LIN {X -0.088,Y -488.926,Z 1104.794,A 0.000,B 0.000,C 90.000,E1 358.969} C_DIS
LIN {X 0.190,Y -496.704,Z 1104.791,A 0.000,B 0.000,C 90.000,E1 358.396} C_DIS
LIN {X -0.080,Y -504.149,Z 1104.788,A 0.000,B 0.000,C 90.000,E1 357.879} C_DIS
LIN {X 0.232,Y -511.620,Z 1104.785,A 0.000,B 0.000,C 90.000,E1 357.249} C_DIS
LIN {X 0.051,Y -516.072,Z 1104.783,A 0.000,B 0.000,C 90.000,E1 356.906} C_DIS
LIN {X 0.077,Y -522.941,Z 1104.779,A 0.000,B 0.000,C 90.000,E1 356.274} C_DIS
LIN {X -0.241,Y -529.630,Z 1104.776,A 0.000,B 0.000,C 90.000,E1 355.641} C_DIS
LIN {X 0.250,Y -535.894,Z 1104.772,A 0.000,B 0.000,C 90.000,E1 354.894} C_DIS
LIN {X -0.207,Y -540.523,Z 1104.769,A 0.000,B 0.000,C 90.000,E1 354.375} C_DIS
LIN {X 0.140,Y -545.729,Z 1104.765,A 0.000,B 0.000,C 90.000,E1 353.628} C_DIS
LIN {X 0.057,Y -550.505,Z 1104.761,A 0.000,B 0.000,C 90.000,E1 352.932} C_DIS
LIN {X 0.201,Y -554.018,Z 1104.758,A 0.000,B 0.000,C 90.000,E1 352.356} C_DIS
LIN {X 0.196,Y -557.831,Z 1104.754,A 0.000,B 0.000,C 90.000,E1 351.659} C_DIS
LIN {X 0.142,Y -561.247,Z 1104.750,A 0.000,B 0.000,C 90.000,E1 350.971} C_DIS
LIN {X 0.135,Y -563.191,Z 1104.748,A 0.000,B 0.000,C 90.000,E1 350.557} C_DIS
LIN {X -0.033,Y -566.692,Z 1104.743,A 0.000,B 0.000,C 90.000,E1 349.746} C_DIS
LIN {X -0.067,Y -569.959,Z 1104.739,A 0.000,B 0.000,C 90.000,E1 348.926} C_DIS
LIN {X 0.014,Y -574.006,Z 1104.732,A 0.000,B 0.000,C 90.000,E1 347.825} C_DIS
LIN {X 0.183,Y -576.822,Z 1104.728,A 0.000,B 0.000,C 90.000,E1 346.992} C_DIS
LIN {X 0.132,Y -581.130,Z 1104.720,A 0.000,B 0.000,C 90.000,E1 345.644} C_DIS
LIN {X 0.059,Y -584.388,Z 1104.714,A 0.000,B 0.000,C 90.000,E1 344.574} C_DIS
LIN {X -0.293,Y -588.324,Z 1104.707,A 0.000,B 0.000,C 90.000,E1 343.268} C_DIS
LIN {X 0.148,Y -592.034,Z 1104.700,A 0.000,B 0.000,C 90.000,E1 341.891} C_DIS
LIN {X -0.166,Y -594.797,Z 1104.694,A 0.000,B 0.000,C 90.000,E1 340.859} C_DIS
LIN {X 0.323,Y -597.309,Z 1104.688,A 0.000,B 0.000,C 90.000,E1 339.752} C_DIS
LIN {X -0.004,Y -600.116,Z 1104.680,A 0.000,B 0.000,C 90.000,E1 338.465} C_DIS
LIN {X 0.086,Y -601.519,Z 1104.676,A 0.000,B 0.000,C 90.000,E1 337.667} C_DIS
LIN {X 0.187,Y -602.833,Z 1104.672,A 0.000,B 0.000,C 90.000,E1 336.869} C_DIS
LIN {X -0.015,Y -603.928,Z 1104.667,A 0.000,B 0.000,C 90.000,E1 336.102} C_DIS
LIN {X 0.042,Y -605.238,Z 1104.661,A 0.000,B 0.000,C 90.000,E1 335.049} C_DIS
LIN {X -0.235,Y -606.531,Z 1104.654,A 0.000,B 0.000,C 90.000,E1 333.768} C_DIS
LIN {X 0.153,Y -607.021,Z 1104.650,A 0.000,B 0.000,C 90.000,E1 332.948} C_DIS
LIN {X 0.284,Y -607.391,Z 1104.646,A 0.000,B 0.000,C 90.000,E1 332.153} C_DIS
LIN {X 0.086,Y -607.526,Z 1104.640,A 0.000,B 0.000,C 90.000,E1 331.129} C_DIS
LIN {X 0.281,Y -607.417,Z 1104.637,A 0.000,B 0.000,C 90.000,E1 330.589} C_DIS
LIN {X -0.151,Y -606.764,Z 1104.631,A 0.000,B 0.000,C 90.000,E1 329.587} C_DIS
LIN {X -0.010,Y -605.795,Z 1104.627,A 0.000,B 0.000,C 90.000,E1 328.791} C_DIS
LIN {X 0.047,Y -604.102,Z 1104.621,A 0.000,B 0.000,C 90.000,E1 327.740} C_DIS
LIN {X -0.032,Y -602.427,Z 1104.616,A 0.000,B 0.000,C 90.000,E1 326.962} C_DIS
LIN {X 0.291,Y -599.833,Z 1104.611,A 0.000,B 0.000,C 90.000,E1 325.881} C_DIS
LIN {X -0.182,Y -596.179,Z 1104.603,A 0.000,B 0.000,C 90.000,E1 324.609} C_DIS
LIN {X -0.016,Y -591.507,Z 1104.594,A 0.000,B 0.000,C 90.000,E1 323.004} C_DIS
LIN {X 0.146,Y -589.181,Z 1104.590,A 0.000,B 0.000,C 90.000,E1 322.190} C_DIS
LIN {X -0.149,Y -585.017,Z 1104.583,A 0.000,B 0.000,C 90.000,E1 320.884} C_DIS
LIN {X -0.050,Y -582.539,Z 1104.578,A 0.000,B 0.000,C 90.000,E1 320.070} C_DIS
LIN {X -0.256,Y -578.919,Z 1104.572,A 0.000,B 0.000,C 90.000,E1 319.013} C_DIS
LIN {X 0.156,Y -575.977,Z 1104.568,A 0.000,B 0.000,C 90.000,E1 318.162} C_DIS
LIN {X -0.276,Y -572.557,Z 1104.563,A 0.000,B 0.000,C 90.000,E1 317.391} C_DIS
LIN {X -0.192,Y -569.234,Z 1104.559,A 0.000,B 0.000,C 90.000,E1 316.701} C_DIS
LIN {X 0.004,Y -566.303,Z 1104.556,A 0.000,B 0.000,C 90.000,E1 316.134} C_DIS
LIN {X 0.024,Y -562.362,Z 1104.552,A 0.000,B 0.000,C 90.000,E1 315.445} C_DIS
LIN {X -0.331,Y -556.410,Z 1104.547,A 0.000,B 0.000,C 90.000,E1 314.514} C_DIS
LIN {X -0.008,Y -551.946,Z 1104.543,A 0.000,B 0.000,C 90.000,E1 313.785} C_DIS
LIN {X -0.110,Y -547.705,Z 1104.539,A 0.000,B 0.000,C 90.000,E1 313.095} C_DIS
LIN {X 0.148,Y -541.824,Z 1104.534,A 0.000,B 0.000,C 90.000,E1 312.081} C_DIS
LIN {X -0.036,Y -538.515,Z 1104.530,A 0.000,B 0.000,C 90.000,E1 311.391} C_DIS
LIN {X 0.013,Y -535.602,Z 1104.525,A 0.000,B 0.000,C 90.000,E1 310.458} C_DIS
LIN {X 0.015,Y -534.100,Z 1104.520,A 0.000,B 0.000,C 90.000,E1 309.600} C_DIS
LIN {X -0.229,Y -533.704,Z 1104.519,A 0.000,B 0.000,C 90.000,E1 309.483} C_DIS
LIN {X -0.071,Y -532.956,Z 1104.516,A 0.000,B 0.000,C 90.000,E1 308.830} C_DIS
LIN {X 0.219,Y -532.151,Z 1104.508,A 0.000,B 0.000,C 90.000,E1 307.363} C_DIS
LIN {X 0.191,Y -532.113,Z 1104.503,A 0.000,B 0.000,C 90.000,E1 306.503} C_DIS
LIN {X 0.171,Y -532.219,Z 1104.500,A 0.000,B 0.000,C 90.000,E1 305.931} C_DIS
LIN {X -0.085,Y -533.150,Z 1104.485,A 0.000,B 0.000,C 90.000,E1 303.372} C_DIS
LIN {X -0.145,Y -534.752,Z 1104.471,A 0.000,B 0.000,C 90.000,E1 300.797} C_DIS
LIN {X 0.175,Y -535.550,Z 1104.465,A 0.000,B 0.000,C 90.000,E1 299.617} C_DIS
LIN {X 0.040,Y -536.287,Z 1104.458,A 0.000,B 0.000,C 90.000,E1 298.487} C_DIS
LIN {X 0.028,Y -537.260,Z 1104.447,A 0.000,B 0.000,C 90.000,E1 296.488} C_DIS
LIN {X -0.142,Y -537.865,Z 1104.439,A 0.000,B 0.000,C 90.000,E1 295.079} C_DIS
LIN {X -0.042,Y -538.253,Z 1104.431,A 0.000,B 0.000,C 90.000,E1 293.643} C_DIS
LIN {X 0.068,Y -538.548,Z 1104.423,A 0.000,B 0.000,C 90.000,E1 292.206} C_DIS
LIN {X -0.246,Y -538.753,Z 1104.417,A 0.000,B 0.000,C 90.000,E1 291.099} C_DIS
LIN {X -0.053,Y -538.752,Z 1104.411,A 0.000,B 0.000,C 90.000,E1 289.939} C_DIS
LIN {X 0.185,Y -538.574,Z 1104.403,A 0.000,B 0.000,C 90.000,E1 288.489} C_DIS
LIN {X -0.096,Y -538.268,Z 1104.395,A 0.000,B 0.000,C 90.000,E1 287.094} C_DIS
LIN {X -0.089,Y -537.971,Z 1104.389,A 0.000,B 0.000,C 90.000,E1 285.953} C_DIS
LIN {X -0.178,Y -537.394,Z 1104.381,A 0.000,B 0.000,C 90.000,E1 284.537} C_DIS
LIN {X -0.211,Y -536.591,Z 1104.371,A 0.000,B 0.000,C 90.000,E1 282.827} C_DIS
LIN {X 0.149,Y -535.751,Z 1104.362,A 0.000,B 0.000,C 90.000,E1 281.074} C_DIS
LIN {X -0.042,Y -534.871,Z 1104.352,A 0.000,B 0.000,C 90.000,E1 279.378} C_DIS
LIN {X 0.096,Y -534.050,Z 1104.343,A 0.000,B 0.000,C 90.000,E1 277.644} C_DIS
LIN {X 0.218,Y -533.208,Z 1104.333,A 0.000,B 0.000,C 90.000,E1 275.910} C_DIS
LIN {X 0.230,Y -532.560,Z 1104.325,A 0.000,B 0.000,C 90.000,E1 274.473} C_DIS
LIN {X 0.201,Y -531.620,Z 1104.314,A 0.000,B 0.000,C 90.000,E1 272.465} C_DIS
LIN {X 0.140,Y -530.818,Z 1104.304,A 0.000,B 0.000,C 90.000,E1 270.745} C_DIS
LIN {X 0.051,Y -529.984,Z 1104.295,A 0.000,B 0.000,C 90.000,E1 269.026} C_DIS
LIN {X -0.025,Y -529.212,Z 1104.287,A 0.000,B 0.000,C 90.000,E1 267.593} C_DIS
LIN {X -0.138,Y -527.983,Z 1104.275,A 0.000,B 0.000,C 90.000,E1 265.584} C_DIS
LIN {X -0.182,Y -527.252,Z 1104.269,A 0.000,B 0.000,C 90.000,E1 264.432} C_DIS
LIN {X -0.249,Y -526.568,Z 1104.264,A 0.000,B 0.000,C 90.000,E1 263.571} C_DIS
LIN {X 0.268,Y -525.419,Z 1104.258,A 0.000,B 0.000,C 90.000,E1 262.356} C_DIS
LIN {X 0.215,Y -523.033,Z 1104.245,A 0.000,B 0.000,C 90.000,E1 260.038} C_DIS
LIN {X 0.253,Y -521.957,Z 1104.238,A 0.000,B 0.000,C 90.000,E1 258.870} C_DIS
LIN {X -0.229,Y -519.974,Z 1104.227,A 0.000,B 0.000,C 90.000,E1 256.881} C_DIS
LIN {X -0.130,Y -518.620,Z 1104.219,A 0.000,B 0.000,C 90.000,E1 255.408} C_DIS
LIN {X 0.072,Y -517.057,Z 1104.211,A 0.000,B 0.000,C 90.000,E1 253.921} C_DIS
LIN {X 0.148,Y -516.161,Z 1104.206,A 0.000,B 0.000,C 90.000,E1 253.032} C_DIS
LIN {X 0.081,Y -514.287,Z 1104.196,A 0.000,B 0.000,C 90.000,E1 251.275} C_DIS
LIN {X -0.084,Y -513.016,Z 1104.190,A 0.000,B 0.000,C 90.000,E1 250.115} C_DIS
LIN {X -0.031,Y -510.937,Z 1104.180,A 0.000,B 0.000,C 90.000,E1 248.337} C_DIS
LIN {X 0.055,Y -509.197,Z 1104.172,A 0.000,B 0.000,C 90.000,E1 246.847} C_DIS
LIN {X 0.101,Y -506.997,Z 1104.163,A 0.000,B 0.000,C 90.000,E1 245.357} C_DIS
LIN {X 0.134,Y -505.675,Z 1104.158,A 0.000,B 0.000,C 90.000,E1 244.460} C_DIS
LIN {X 0.235,Y -503.739,Z 1104.152,A 0.000,B 0.000,C 90.000,E1 243.256} C_DIS
LIN {X -0.232,Y -500.810,Z 1104.142,A 0.000,B 0.000,C 90.000,E1 241.513} C_DIS
LIN {X 0.155,Y -497.771,Z 1104.132,A 0.000,B 0.000,C 90.000,E1 239.665} C_DIS
LIN {X 0.174,Y -495.736,Z 1104.125,A 0.000,B 0.000,C 90.000,E1 238.456} C_DIS
LIN {X 0.275,Y -492.520,Z 1104.115,A 0.000,B 0.000,C 90.000,E1 236.628} C_DIS
LIN {X -0.204,Y -490.375,Z 1104.108,A 0.000,B 0.000,C 90.000,E1 235.468} C_DIS
LIN {X 0.081,Y -487.511,Z 1104.100,A 0.000,B 0.000,C 90.000,E1 233.909} C_DIS
LIN {X -0.075,Y -484.603,Z 1104.091,A 0.000,B 0.000,C 90.000,E1 232.396} C_DIS
LIN {X 0.017,Y -481.539,Z 1104.083,A 0.000,B 0.000,C 90.000,E1 230.848} C_DIS
LIN {X -0.044,Y -477.231,Z 1104.071,A 0.000,B 0.000,C 90.000,E1 228.690} C_DIS
LIN {X -0.176,Y -472.439,Z 1104.057,A 0.000,B 0.000,C 90.000,E1 226.215} C_DIS
LIN {X -0.057,Y -469.619,Z 1104.048,A 0.000,B 0.000,C 90.000,E1 224.636} C_DIS
LIN {X -0.067,Y -467.362,Z 1104.041,A 0.000,B 0.000,C 90.000,E1 223.380} C_DIS
LIN {X 0.104,Y -463.361,Z 1104.029,A 0.000,B 0.000,C 90.000,E1 221.148} C_DIS
LIN {X 0.218,Y -459.609,Z 1104.016,A 0.000,B 0.000,C 90.000,E1 218.910} C_DIS
LIN {X -0.068,Y -456.459,Z 1104.006,A 0.000,B 0.000,C 90.000,E1 217.030} C_DIS
LIN {X -0.060,Y -453.498,Z 1103.995,A 0.000,B 0.000,C 90.000,E1 215.105} C_DIS
LIN {X 0.069,Y -450.030,Z 1103.983,A 0.000,B 0.000,C 90.000,E1 212.832} C_DIS
LIN {X 0.169,Y -447.237,Z 1103.972,A 0.000,B 0.000,C 90.000,E1 210.875} C_DIS
LIN {X -0.014,Y -443.021,Z 1103.954,A 0.000,B 0.000,C 90.000,E1 207.641} C_DIS
LIN {X 0.091,Y -440.560,Z 1103.941,A 0.000,B 0.000,C 90.000,E1 205.335} C_DIS
LIN {X 0.076,Y -439.566,Z 1103.932,A 0.000,B 0.000,C 90.000,E1 203.695} C_DIS
LIN {X 0.024,Y -439.516,Z 1103.924,A 0.000,B 0.000,C 90.000,E1 202.386} C_DIS
LIN {X -0.037,Y -440.005,Z 1103.919,A 0.000,B 0.000,C 90.000,E1 201.408} C_DIS
LIN {X 0.065,Y -440.657,Z 1103.915,A 0.000,B 0.000,C 90.000,E1 200.737} C_DIS
LIN {X 0.174,Y -441.671,Z 1103.912,A 0.000,B 0.000,C 90.000,E1 200.066} C_DIS
LIN {X 0.142,Y -443.785,Z 1103.906,A 0.000,B 0.000,C 90.000,E1 199.087} C_DIS
LIN {X -0.010,Y -446.435,Z 1103.901,A 0.000,B 0.000,C 90.000,E1 198.127} C_DIS
LIN {X 0.040,Y -451.871,Z 1103.892,A 0.000,B 0.000,C 90.000,E1 196.496} C_DIS
LIN {X -0.008,Y -464.587,Z 1103.874,A 0.000,B 0.000,C 90.000,E1 193.300} C_DIS
LIN {X 0.197,Y -476.298,Z 1103.859,A 0.000,B 0.000,C 90.000,E1 190.602} C_DIS
LIN {X -0.165,Y -483.419,Z 1103.850,A 0.000,B 0.000,C 90.000,E1 189.095} C_DIS
LIN {X -0.062,Y -489.809,Z 1103.843,A 0.000,B 0.000,C 90.000,E1 187.701} C_DIS
LIN {X -0.243,Y -496.743,Z 1103.834,A 0.000,B 0.000,C 90.000,E1 186.201} C_DIS
LIN {X 0.077,Y -504.800,Z 1103.824,A 0.000,B 0.000,C 90.000,E1 184.359} C_DIS
LIN {X 0.126,Y -511.555,Z 1103.816,A 0.000,B 0.000,C 90.000,E1 182.865} C_DIS
LIN {X -0.079,Y -520.276,Z 1103.805,A 0.000,B 0.000,C 90.000,E1 180.974} C_DIS
LIN {X 0.222,Y -527.050,Z 1103.797,A 0.000,B 0.000,C 90.000,E1 179.484} C_DIS
LIN {X 0.135,Y -533.740,Z 1103.789,A 0.000,B 0.000,C 90.000,E1 178.051} C_DIS
LIN {X -0.103,Y -539.767,Z 1103.782,A 0.000,B 0.000,C 90.000,E1 176.788} C_DIS
LIN {X 0.007,Y -545.093,Z 1103.776,A 0.000,B 0.000,C 90.000,E1 175.641} C_DIS
LIN {X -0.169,Y -552.915,Z 1103.766,A 0.000,B 0.000,C 90.000,E1 173.970} C_DIS
LIN {X 0.065,Y -560.117,Z 1103.758,A 0.000,B 0.000,C 90.000,E1 172.413} C_DIS
LIN {X -0.052,Y -565.284,Z 1103.752,A 0.000,B 0.000,C 90.000,E1 171.319} C_DIS
LIN {X -0.162,Y -570.987,Z 1103.745,A 0.000,B 0.000,C 90.000,E1 170.095} C_DIS
LIN {X -0.199,Y -578.362,Z 1103.736,A 0.000,B 0.000,C 90.000,E1 168.465} C_DIS
LIN {X -0.218,Y -584.227,Z 1103.728,A 0.000,B 0.000,C 90.000,E1 167.117} C_DIS
LIN {X 0.320,Y -588.658,Z 1103.722,A 0.000,B 0.000,C 90.000,E1 165.992} C_DIS
LIN {X 0.206,Y -592.896,Z 1103.716,A 0.000,B 0.000,C 90.000,E1 164.936} C_DIS
LIN {X -0.276,Y -596.934,Z 1103.711,A 0.000,B 0.000,C 90.000,E1 163.921} C_DIS
LIN {X 0.044,Y -600.692,Z 1103.705,A 0.000,B 0.000,C 90.000,E1 162.834} C_DIS
LIN {X 0.240,Y -604.257,Z 1103.699,A 0.000,B 0.000,C 90.000,E1 161.764} C_DIS
LIN {X -0.180,Y -608.308,Z 1103.692,A 0.000,B 0.000,C 90.000,E1 160.496} C_DIS
LIN {X -0.062,Y -611.408,Z 1103.686,A 0.000,B 0.000,C 90.000,E1 159.444} C_DIS
LIN {X -0.114,Y -614.384,Z 1103.680,A 0.000,B 0.000,C 90.000,E1 158.411} C_DIS
LIN {X 0.073,Y -617.924,Z 1103.673,A 0.000,B 0.000,C 90.000,E1 157.102} C_DIS
LIN {X 0.320,Y -622.024,Z 1103.664,A 0.000,B 0.000,C 90.000,E1 155.537} C_DIS
LIN {X 0.079,Y -625.940,Z 1103.656,A 0.000,B 0.000,C 90.000,E1 154.024} C_DIS
LIN {X 0.161,Y -629.006,Z 1103.649,A 0.000,B 0.000,C 90.000,E1 152.743} C_DIS
LIN {X -0.238,Y -632.386,Z 1103.640,A 0.000,B 0.000,C 90.000,E1 151.257} C_DIS
LIN {X -0.271,Y -635.740,Z 1103.632,A 0.000,B 0.000,C 90.000,E1 149.744} C_DIS
LIN {X 0.042,Y -638.341,Z 1103.625,A 0.000,B 0.000,C 90.000,E1 148.456} C_DIS
LIN {X 0.064,Y -640.833,Z 1103.618,A 0.000,B 0.000,C 90.000,E1 147.199} C_DIS
LIN {X -0.077,Y -643.237,Z 1103.611,A 0.000,B 0.000,C 90.000,E1 145.960} C_DIS
LIN {X -0.227,Y -645.049,Z 1103.605,A 0.000,B 0.000,C 90.000,E1 144.975} C_DIS
LIN {X -0.018,Y -647.746,Z 1103.597,A 0.000,B 0.000,C 90.000,E1 143.463} C_DIS
LIN {X -0.142,Y -650.395,Z 1103.589,A 0.000,B 0.000,C 90.000,E1 141.984} C_DIS
LIN {X 0.105,Y -653.631,Z 1103.579,A 0.000,B 0.000,C 90.000,E1 140.231} C_DIS
LIN {X 0.306,Y -657.423,Z 1103.568,A 0.000,B 0.000,C 90.000,E1 138.243} C_DIS
LIN {X 0.170,Y -660.396,Z 1103.560,A 0.000,B 0.000,C 90.000,E1 136.782} C_DIS
LIN {X 0.033,Y -665.717,Z 1103.547,A 0.000,B 0.000,C 90.000,E1 134.352} C_DIS
LIN {X 0.081,Y -670.402,Z 1103.536,A 0.000,B 0.000,C 90.000,E1 132.405} C_DIS
LIN {X -0.296,Y -674.041,Z 1103.528,A 0.000,B 0.000,C 90.000,E1 130.987} C_DIS
LIN {X -0.025,Y -677.589,Z 1103.520,A 0.000,B 0.000,C 90.000,E1 129.519} C_DIS
LIN {X 0.356,Y -681.922,Z 1103.510,A 0.000,B 0.000,C 90.000,E1 127.810} C_DIS
LIN {X -0.206,Y -684.985,Z 1103.504,A 0.000,B 0.000,C 90.000,E1 126.664} C_DIS
LIN {X -0.137,Y -688.563,Z 1103.496,A 0.000,B 0.000,C 90.000,E1 125.231} C_DIS
LIN {X -0.049,Y -691.400,Z 1103.489,A 0.000,B 0.000,C 90.000,E1 124.040} C_DIS
LIN {X -0.302,Y -694.311,Z 1103.483,A 0.000,B 0.000,C 90.000,E1 122.880} C_DIS
LIN {X -0.162,Y -696.602,Z 1103.477,A 0.000,B 0.000,C 90.000,E1 121.926} C_DIS
LIN {X -0.357,Y -698.662,Z 1103.472,A 0.000,B 0.000,C 90.000,E1 121.003} C_DIS
LIN {X -0.168,Y -700.440,Z 1103.467,A 0.000,B 0.000,C 90.000,E1 120.050} C_DIS
LIN {X -0.042,Y -702.354,Z 1103.460,A 0.000,B 0.000,C 90.000,E1 118.871} C_DIS
LIN {X 0.121,Y -703.558,Z 1103.455,A 0.000,B 0.000,C 90.000,E1 117.924} C_DIS
LIN {X -0.273,Y -704.299,Z 1103.451,A 0.000,B 0.000,C 90.000,E1 117.257} C_DIS
LIN {X -0.124,Y -705.370,Z 1103.444,A 0.000,B 0.000,C 90.000,E1 115.848} C_DIS
LIN {X -0.194,Y -705.737,Z 1103.440,A 0.000,B 0.000,C 90.000,E1 115.155} C_DIS
LIN {X 0.387,Y -705.696,Z 1103.437,A 0.000,B 0.000,C 90.000,E1 114.643} C_DIS
LIN {X -0.258,Y -705.486,Z 1103.436,A 0.000,B 0.000,C 90.000,E1 114.463} C_DIS
LIN {X 0.319,Y -704.770,Z 1103.433,A 0.000,B 0.000,C 90.000,E1 113.951} C_DIS
LIN {X -0.040,Y -703.023,Z 1103.431,A 0.000,B 0.000,C 90.000,E1 113.515} C_DIS
LIN {X 0.239,Y -701.954,Z 1103.429,A 0.000,B 0.000,C 90.000,E1 113.259} C_DIS
LIN {X -0.033,Y -698.059,Z 1103.427,A 0.000,B 0.000,C 90.000,E1 112.823} C_DIS
LIN {X 0.096,Y -696.956,Z 1103.426,A 0.000,B 0.000,C 90.000,E1 112.695} C_DIS
LIN {X -0.042,Y -695.323,Z 1103.426,A 0.000,B 0.000,C 90.000,E1 112.589} C_DIS
LIN {X -0.005,Y -690.723,Z 1103.424,A 0.000,B 0.000,C 90.000,E1 112.386} C_DIS
LIN {X -0.108,Y -687.387,Z 1103.424,A 0.000,B 0.000,C 90.000,E1 112.259} C_DIS
LIN {X -0.283,Y -685.495,Z 1103.423,A 0.000,B 0.000,C 90.000,E1 112.206} C_DIS
LIN {X -0.053,Y -683.590,Z 1103.423,A 0.000,B 0.000,C 90.000,E1 112.153} C_DIS
LIN {X -0.199,Y -675.939,Z 1103.423,A 0.000,B 0.000,C 90.000,E1 112.078} C_DIS
LIN {X -0.225,Y -604.098,Z 1103.423,A 0.000,B 0.000,C 90.000,E1 112.078} C_DIS
LIN {X 0.135,Y -600.461,Z 1103.422,A 0.000,B 0.000,C 90.000,E1 111.844} C_DIS
LIN {X 0.160,Y -596.106,Z 1103.420,A 0.000,B 0.000,C 90.000,E1 111.535} C_DIS
LIN {X -0.062,Y -578.609,Z 1103.411,A 0.000,B 0.000,C 90.000,E1 110.066} C_DIS
LIN {X -0.014,Y -574.362,Z 1103.410,A 0.000,B 0.000,C 90.000,E1 109.704} C_DIS
LIN {X -0.171,Y -568.294,Z 1103.407,A 0.000,B 0.000,C 90.000,E1 109.268} C_DIS
LIN {X 0.173,Y -560.101,Z 1103.404,A 0.000,B 0.000,C 90.000,E1 108.725} C_DIS
LIN {X 0.117,Y -553.768,Z 1103.402,A 0.000,B 0.000,C 90.000,E1 108.362} C_DIS
LIN {X 0.221,Y -549.835,Z 1103.401,A 0.000,B 0.000,C 90.000,E1 108.055} C_DIS
LIN {X 0.135,Y -548.522,Z 1103.399,A 0.000,B 0.000,C 90.000,E1 107.873} C_DIS
LIN {X 0.094,Y -548.497,Z 1103.399,A 0.000,B 0.000,C 90.000,E1 107.873} C_DIS
LIN {X 0.224,Y -548.201,Z 1103.398,A 0.000,B 0.000,C 90.000,E1 107.583} C_DIS
LIN {X 0.264,Y -548.501,Z 1103.393,A 0.000,B 0.000,C 90.000,E1 106.677} C_DIS
LIN {X -0.234,Y -550.066,Z 1103.380,A 0.000,B 0.000,C 90.000,E1 104.481} C_DIS
LIN {X -0.284,Y -551.856,Z 1103.368,A 0.000,B 0.000,C 90.000,E1 102.243} C_DIS
LIN {X -0.107,Y -553.448,Z 1103.359,A 0.000,B 0.000,C 90.000,E1 100.546} C_DIS
LIN {X 0.126,Y -555.451,Z 1103.348,A 0.000,B 0.000,C 90.000,E1 98.568} C_DIS
LIN {X 0.060,Y -556.875,Z 1103.340,A 0.000,B 0.000,C 90.000,E1 97.182} C_DIS
LIN {X -0.108,Y -558.046,Z 1103.334,A 0.000,B 0.000,C 90.000,E1 96.087} C_DIS
LIN {X -0.260,Y -559.127,Z 1103.328,A 0.000,B 0.000,C 90.000,E1 94.992} C_DIS
LIN {X 0.241,Y -560.227,Z 1103.320,A 0.000,B 0.000,C 90.000,E1 93.555} C_DIS
LIN {X 0.167,Y -561.129,Z 1103.312,A 0.000,B 0.000,C 90.000,E1 92.178} C_DIS
LIN {X 0.206,Y -562.026,Z 1103.303,A 0.000,B 0.000,C 90.000,E1 90.516} C_DIS
LIN {X -0.054,Y -562.417,Z 1103.298,A 0.000,B 0.000,C 90.000,E1 89.714} C_DIS
LIN {X -0.108,Y -563.095,Z 1103.291,A 0.000,B 0.000,C 90.000,E1 88.339} C_DIS
LIN {X -0.006,Y -563.848,Z 1103.282,A 0.000,B 0.000,C 90.000,E1 86.674} C_DIS
LIN {X 0.121,Y -564.536,Z 1103.272,A 0.000,B 0.000,C 90.000,E1 85.008} C_DIS
LIN {X 0.154,Y -565.074,Z 1103.265,A 0.000,B 0.000,C 90.000,E1 83.628} C_DIS
LIN {X -0.141,Y -565.651,Z 1103.256,A 0.000,B 0.000,C 90.000,E1 82.008} C_DIS
LIN {X -0.035,Y -566.092,Z 1103.248,A 0.000,B 0.000,C 90.000,E1 80.622} C_DIS
LIN {X -0.224,Y -566.822,Z 1103.239,A 0.000,B 0.000,C 90.000,E1 78.993} C_DIS
LIN {X -0.113,Y -567.727,Z 1103.228,A 0.000,B 0.000,C 90.000,E1 77.061} C_DIS
LIN {X -0.006,Y -568.141,Z 1103.224,A 0.000,B 0.000,C 90.000,E1 76.228} C_DIS
LIN {X -0.279,Y -569.258,Z 1103.213,A 0.000,B 0.000,C 90.000,E1 74.338} C_DIS
LIN {X -0.046,Y -570.883,Z 1103.201,A 0.000,B 0.000,C 90.000,E1 72.127} C_DIS
LIN {X -0.121,Y -572.191,Z 1103.192,A 0.000,B 0.000,C 90.000,E1 70.496} C_DIS
LIN {X -0.150,Y -573.922,Z 1103.181,A 0.000,B 0.000,C 90.000,E1 68.592} C_DIS
LIN {X 0.085,Y -575.573,Z 1103.170,A 0.000,B 0.000,C 90.000,E1 66.666} C_DIS
LIN {X -0.173,Y -577.120,Z 1103.160,A 0.000,B 0.000,C 90.000,E1 64.793} C_DIS
LIN {X 0.093,Y -578.465,Z 1103.149,A 0.000,B 0.000,C 90.000,E1 62.871} C_DIS
LIN {X 0.301,Y -579.266,Z 1103.143,A 0.000,B 0.000,C 90.000,E1 61.769} C_DIS
LIN {X -0.273,Y -580.257,Z 1103.134,A 0.000,B 0.000,C 90.000,E1 60.205} C_DIS
LIN {X 0.097,Y -581.024,Z 1103.127,A 0.000,B 0.000,C 90.000,E1 58.820} C_DIS
LIN {X 0.286,Y -581.758,Z 1103.119,A 0.000,B 0.000,C 90.000,E1 57.454} C_DIS
LIN {X 0.033,Y -582.759,Z 1103.109,A 0.000,B 0.000,C 90.000,E1 55.595} C_DIS
LIN {X 0.132,Y -583.555,Z 1103.099,A 0.000,B 0.000,C 90.000,E1 53.703} C_DIS
LIN {X -0.058,Y -584.122,Z 1103.089,A 0.000,B 0.000,C 90.000,E1 52.110} C_DIS
LIN {X 0.035,Y -584.329,Z 1103.085,A 0.000,B 0.000,C 90.000,E1 51.295} C_DIS
LIN {X -0.060,Y -584.325,Z 1103.079,A 0.000,B 0.000,C 90.000,E1 50.231} C_DIS
LIN {X 0.142,Y -584.187,Z 1103.073,A 0.000,B 0.000,C 90.000,E1 49.138} C_DIS
LIN {X 0.139,Y -583.893,Z 1103.066,A 0.000,B 0.000,C 90.000,E1 47.796} C_DIS
LIN {X 0.082,Y -583.452,Z 1103.058,A 0.000,B 0.000,C 90.000,E1 46.458} C_DIS
LIN {X 0.011,Y -582.722,Z 1103.051,A 0.000,B 0.000,C 90.000,E1 45.121} C_DIS
LIN {X 0.194,Y -582.030,Z 1103.045,A 0.000,B 0.000,C 90.000,E1 44.028} C_DIS
LIN {X -0.051,Y -580.942,Z 1103.039,A 0.000,B 0.000,C 90.000,E1 42.975} C_DIS
LIN {X -0.008,Y -580.031,Z 1103.034,A 0.000,B 0.000,C 90.000,E1 42.162} C_DIS
LIN {X -0.139,Y -578.249,Z 1103.027,A 0.000,B 0.000,C 90.000,E1 40.825} C_DIS
LIN {X -0.114,Y -577.041,Z 1103.022,A 0.000,B 0.000,C 90.000,E1 40.011} C_DIS
LIN {X 0.053,Y -575.199,Z 1103.016,A 0.000,B 0.000,C 90.000,E1 38.910} C_DIS
LIN {X -0.116,Y -572.378,Z 1103.009,A 0.000,B 0.000,C 90.000,E1 37.569} C_DIS
LIN {X -0.045,Y -570.391,Z 1103.004,A 0.000,B 0.000,C 90.000,E1 36.744} C_DIS
LIN {X -0.109,Y -568.042,Z 1103.000,A 0.000,B 0.000,C 90.000,E1 35.931} C_DIS
LIN {X -0.192,Y -566.293,Z 1102.997,A 0.000,B 0.000,C 90.000,E1 35.391} C_DIS
LIN {X -0.060,Y -562.298,Z 1102.990,A 0.000,B 0.000,C 90.000,E1 34.278} C_DIS
LIN {X -0.076,Y -558.835,Z 1102.986,A 0.000,B 0.000,C 90.000,E1 33.452} C_DIS
LIN {X -0.019,Y -555.675,Z 1102.982,A 0.000,B 0.000,C 90.000,E1 32.752} C_DIS
LIN {X -0.118,Y -551.667,Z 1102.977,A 0.000,B 0.000,C 90.000,E1 31.926} C_DIS
LIN {X -0.046,Y -545.733,Z 1102.971,A 0.000,B 0.000,C 90.000,E1 30.797} C_DIS
LIN {X -0.191,Y -538.358,Z 1102.964,A 0.000,B 0.000,C 90.000,E1 29.539} C_DIS
LIN {X -0.145,Y -533.758,Z 1102.960,A 0.000,B 0.000,C 90.000,E1 28.821} C_DIS
LIN {X -0.286,Y -527.834,Z 1102.955,A 0.000,B 0.000,C 90.000,E1 27.975} C_DIS
LIN {X 0.131,Y -522.304,Z 1102.951,A 0.000,B 0.000,C 90.000,E1 27.206} C_DIS
LIN {X 0.229,Y -517.599,Z 1102.948,A 0.000,B 0.000,C 90.000,E1 26.616} C_DIS
LIN {X 0.024,Y -512.510,Z 1102.945,A 0.000,B 0.000,C 90.000,E1 26.052} C_DIS
LIN {X 0.218,Y -507.351,Z 1102.942,A 0.000,B 0.000,C 90.000,E1 25.463} C_DIS
LIN {X -0.203,Y -497.889,Z 1102.936,A 0.000,B 0.000,C 90.000,E1 24.515} C_DIS
LIN {X 0.096,Y -489.491,Z 1102.932,A 0.000,B 0.000,C 90.000,E1 23.643} C_DIS
LIN {X -0.200,Y -477.911,Z 1102.925,A 0.000,B 0.000,C 90.000,E1 22.589} C_DIS
LIN {X -0.152,Y -465.952,Z 1102.920,A 0.000,B 0.000,C 90.000,E1 21.535} C_DIS
LIN {X -0.015,Y -449.463,Z 1102.911,A 0.000,B 0.000,C 90.000,E1 20.066} C_DIS
LIN {X 0.040,Y -432.026,Z 1102.902,A 0.000,B 0.000,C 90.000,E1 18.417} C_DIS
LIN {X -0.017,Y -419.346,Z 1102.895,A 0.000,B 0.000,C 90.000,E1 17.094} C_DIS
LIN {X -0.114,Y -409.970,Z 1102.889,A 0.000,B 0.000,C 90.000,E1 16.024} C_DIS
LIN {X 0.114,Y -401.003,Z 1102.883,A 0.000,B 0.000,C 90.000,E1 14.828} C_DIS
LIN {X -0.138,Y -397.567,Z 1102.880,A 0.000,B 0.000,C 90.000,E1 14.356} C_DIS
LIN {X -0.065,Y -395.396,Z 1102.877,A 0.000,B 0.000,C 90.000,E1 13.939} C_DIS
LIN {X -0.049,Y -393.112,Z 1102.874,A 0.000,B 0.000,C 90.000,E1 13.355} C_DIS
LIN {X -0.008,Y -392.223,Z 1102.871,A 0.000,B 0.000,C 90.000,E1 12.827} C_DIS
LIN {X 0.033,Y -392.155,Z 1102.867,A 0.000,B 0.000,C 90.000,E1 12.119} C_DIS
LIN {X -0.060,Y -392.875,Z 1102.863,A 0.000,B 0.000,C 90.000,E1 11.422} C_DIS
LIN {X 0.203,Y -395.982,Z 1102.854,A 0.000,B 0.000,C 90.000,E1 9.613} C_DIS
LIN {X 0.091,Y -399.000,Z 1102.846,A 0.000,B 0.000,C 90.000,E1 8.219} C_DIS
LIN {X -0.031,Y -402.438,Z 1102.838,A 0.000,B 0.000,C 90.000,E1 6.834} C_DIS
LIN {X -0.102,Y -405.822,Z 1102.830,A 0.000,B 0.000,C 90.000,E1 5.448} C_DIS
LIN {X -0.141,Y -406.876,Z 1102.828,A 0.000,B 0.000,C 90.000,E1 5.106} C_DIS
LIN {X -0.118,Y -410.073,Z 1102.824,A 0.000,B 0.000,C 90.000,E1 4.416} C_DIS
LIN {X 0.171,Y -411.750,Z 1102.823,A 0.000,B 0.000,C 90.000,E1 4.131} C_DIS
LIN {X 0.176,Y -416.475,Z 1102.821,A 0.000,B 0.000,C 90.000,E1 3.669} C_DIS
LIN {X -0.044,Y -425.708,Z 1102.817,A 0.000,B 0.000,C 90.000,E1 3.037} C_DIS
LIN {X -0.108,Y -445.427,Z 1102.810,A 0.000,B 0.000,C 90.000,E1 1.718} C_DIS
LIN {X 0.087,Y -461.885,Z 1102.804,A 0.000,B 0.000,C 90.000,E1 0.630} C_DIS
LIN {X -0.191,Y -476.994,Z 1102.798,A 0.000,B 0.000,C 90.000,E1 359.714} C_DIS
LIN {X -0.173,Y -486.631,Z 1102.795,A 0.000,B 0.000,C 90.000,E1 359.083} C_DIS
LIN {X 0.077,Y -492.969,Z 1102.792,A 0.000,B 0.000,C 90.000,E1 358.625} C_DIS
LIN {X 0.218,Y -499.242,Z 1102.790,A 0.000,B 0.000,C 90.000,E1 358.167} C_DIS
LIN {X -0.211,Y -503.845,Z 1102.788,A 0.000,B 0.000,C 90.000,E1 357.879} C_DIS
LIN {X -0.242,Y -511.147,Z 1102.785,A 0.000,B 0.000,C 90.000,E1 357.306} C_DIS
LIN {X 0.083,Y -516.957,Z 1102.782,A 0.000,B 0.000,C 90.000,E1 356.788} C_DIS
LIN {X 0.013,Y -523.877,Z 1102.779,A 0.000,B 0.000,C 90.000,E1 356.159} C_DIS
LIN {X -0.153,Y -529.313,Z 1102.776,A 0.000,B 0.000,C 90.000,E1 355.641} C_DIS
LIN {X -0.075,Y -535.532,Z 1102.772,A 0.000,B 0.000,C 90.000,E1 354.951} C_DIS
LIN {X -0.205,Y -541.260,Z 1102.768,A 0.000,B 0.000,C 90.000,E1 354.261} C_DIS
LIN {X -0.131,Y -545.470,Z 1102.765,A 0.000,B 0.000,C 90.000,E1 353.685} C_DIS
LIN {X -0.218,Y -550.316,Z 1102.761,A 0.000,B 0.000,C 90.000,E1 352.989} C_DIS
LIN {X -0.077,Y -553.863,Z 1102.758,A 0.000,B 0.000,C 90.000,E1 352.413} C_DIS
LIN {X -0.163,Y -557.735,Z 1102.754,A 0.000,B 0.000,C 90.000,E1 351.724} C_DIS
LIN {X -0.139,Y -561.209,Z 1102.750,A 0.000,B 0.000,C 90.000,E1 351.027} C_DIS
LIN {X -0.082,Y -564.385,Z 1102.746,A 0.000,B 0.000,C 90.000,E1 350.330} C_DIS
LIN {X -0.142,Y -567.867,Z 1102.742,A 0.000,B 0.000,C 90.000,E1 349.511} C_DIS
LIN {X -0.274,Y -571.080,Z 1102.737,A 0.000,B 0.000,C 90.000,E1 348.701} C_DIS
LIN {X -0.067,Y -575.107,Z 1102.731,A 0.000,B 0.000,C 90.000,E1 347.589} C_DIS
LIN {X -0.233,Y -578.724,Z 1102.725,A 0.000,B 0.000,C 90.000,E1 346.520} C_DIS
LIN {X -0.257,Y -582.961,Z 1102.718,A 0.000,B 0.000,C 90.000,E1 345.172} C_DIS
LIN {X -0.307,Y -586.194,Z 1102.712,A 0.000,B 0.000,C 90.000,E1 344.102} C_DIS
LIN {X 0.099,Y -590.087,Z 1102.704,A 0.000,B 0.000,C 90.000,E1 342.725} C_DIS
LIN {X 0.325,Y -593.054,Z 1102.698,A 0.000,B 0.000,C 90.000,E1 341.638} C_DIS
LIN {X 0.032,Y -595.797,Z 1102.692,A 0.000,B 0.000,C 90.000,E1 340.604} C_DIS
LIN {X -0.226,Y -598.245,Z 1102.686,A 0.000,B 0.000,C 90.000,E1 339.571} C_DIS
LIN {X 0.016,Y -601.019,Z 1102.679,A 0.000,B 0.000,C 90.000,E1 338.230} C_DIS
LIN {X -0.034,Y -603.262,Z 1102.672,A 0.000,B 0.000,C 90.000,E1 336.922} C_DIS
LIN {X 0.016,Y -604.703,Z 1102.666,A 0.000,B 0.000,C 90.000,E1 335.869} C_DIS
LIN {X -0.162,Y -605.744,Z 1102.662,A 0.000,B 0.000,C 90.000,E1 335.101} C_DIS
LIN {X 0.121,Y -607.047,Z 1102.654,A 0.000,B 0.000,C 90.000,E1 333.768} C_DIS
LIN {X 0.022,Y -607.475,Z 1102.651,A 0.000,B 0.000,C 90.000,E1 333.256} C_DIS
LIN {X -0.170,Y -608.001,Z 1102.646,A 0.000,B 0.000,C 90.000,E1 332.231} C_DIS
LIN {X -0.070,Y -608.217,Z 1102.640,A 0.000,B 0.000,C 90.000,E1 331.179} C_DIS
LIN {X -0.166,Y -608.231,Z 1102.637,A 0.000,B 0.000,C 90.000,E1 330.667} C_DIS
LIN {X -0.067,Y -607.653,Z 1102.631,A 0.000,B 0.000,C 90.000,E1 329.616} C_DIS
LIN {X 0.133,Y -607.106,Z 1102.628,A 0.000,B 0.000,C 90.000,E1 329.076} C_DIS
LIN {X -0.245,Y -606.032,Z 1102.624,A 0.000,B 0.000,C 90.000,E1 328.329} C_DIS
LIN {X -0.119,Y -604.767,Z 1102.620,A 0.000,B 0.000,C 90.000,E1 327.533} C_DIS
LIN {X -0.189,Y -603.121,Z 1102.615,A 0.000,B 0.000,C 90.000,E1 326.755} C_DIS
LIN {X -0.104,Y -601.295,Z 1102.611,A 0.000,B 0.000,C 90.000,E1 325.960} C_DIS
LIN {X 0.040,Y -598.550,Z 1102.605,A 0.000,B 0.000,C 90.000,E1 324.895} C_DIS
LIN {X -0.080,Y -596.411,Z 1102.601,A 0.000,B 0.000,C 90.000,E1 324.116} C_DIS
LIN {X 0.226,Y -592.803,Z 1102.593,A 0.000,B 0.000,C 90.000,E1 322.763} C_DIS
LIN {X -0.384,Y -591.999,Z 1102.592,A 0.000,B 0.000,C 90.000,E1 322.557} C_DIS
LIN {X 0.044,Y -590.666,Z 1102.589,A 0.000,B 0.000,C 90.000,E1 321.984} C_DIS
LIN {X 0.143,Y -586.901,Z 1102.581,A 0.000,B 0.000,C 90.000,E1 320.642} C_DIS
LIN {X 0.001,Y -583.827,Z 1102.576,A 0.000,B 0.000,C 90.000,E1 319.585} C_DIS
LIN {X -0.181,Y -580.540,Z 1102.570,A 0.000,B 0.000,C 90.000,E1 318.528} C_DIS
LIN {X -0.135,Y -577.786,Z 1102.565,A 0.000,B 0.000,C 90.000,E1 317.715} C_DIS
LIN {X 0.124,Y -575.569,Z 1102.562,A 0.000,B 0.000,C 90.000,E1 317.148} C_DIS
LIN {X -0.313,Y -571.958,Z 1102.557,A 0.000,B 0.000,C 90.000,E1 316.377} C_DIS
LIN {X -0.094,Y -569.153,Z 1102.554,A 0.000,B 0.000,C 90.000,E1 315.810} C_DIS
LIN {X -0.280,Y -562.324,Z 1102.548,A 0.000,B 0.000,C 90.000,E1 314.595} C_DIS
LIN {X 0.326,Y -557.529,Z 1102.543,A 0.000,B 0.000,C 90.000,E1 313.704} C_DIS
LIN {X 0.084,Y -552.637,Z 1102.538,A 0.000,B 0.000,C 90.000,E1 312.894} C_DIS
LIN {X 0.068,Y -545.027,Z 1102.531,A 0.000,B 0.000,C 90.000,E1 311.634} C_DIS
LIN {X 0.079,Y -541.878,Z 1102.528,A 0.000,B 0.000,C 90.000,E1 311.067} C_DIS
LIN {X -0.087,Y -539.493,Z 1102.525,A 0.000,B 0.000,C 90.000,E1 310.539} C_DIS
LIN {X -0.055,Y -537.641,Z 1102.522,A 0.000,B 0.000,C 90.000,E1 309.967} C_DIS
LIN {X 0.300,Y -536.806,Z 1102.521,A 0.000,B 0.000,C 90.000,E1 309.644} C_DIS
LIN {X -0.095,Y -534.593,Z 1102.514,A 0.000,B 0.000,C 90.000,E1 308.543} C_DIS
LIN {X -0.094,Y -534.659,Z 1102.513,A 0.000,B 0.000,C 90.000,E1 308.257} C_DIS
LIN {X -0.050,Y -533.813,Z 1102.509,A 0.000,B 0.000,C 90.000,E1 307.684} C_DIS
LIN {X 0.056,Y -533.695,Z 1102.508,A 0.000,B 0.000,C 90.000,E1 307.397} C_DIS
LIN {X 0.054,Y -533.351,Z 1102.506,A 0.000,B 0.000,C 90.000,E1 307.111} C_DIS
LIN {X -0.264,Y -533.344,Z 1102.503,A 0.000,B 0.000,C 90.000,E1 306.583} C_DIS
LIN {X -0.268,Y -533.043,Z 1102.502,A 0.000,B 0.000,C 90.000,E1 306.297} C_DIS
LIN {X 0.154,Y -533.053,Z 1102.498,A 0.000,B 0.000,C 90.000,E1 305.678} C_DIS
LIN {X 0.142,Y -532.987,Z 1102.495,A 0.000,B 0.000,C 90.000,E1 305.105} C_DIS
LIN {X -0.075,Y -533.758,Z 1102.482,A 0.000,B 0.000,C 90.000,E1 302.832} C_DIS
LIN {X -0.116,Y -535.377,Z 1102.468,A 0.000,B 0.000,C 90.000,E1 300.256} C_DIS
LIN {X -0.093,Y -536.453,Z 1102.458,A 0.000,B 0.000,C 90.000,E1 298.537} C_DIS
LIN {X -0.109,Y -537.433,Z 1102.447,A 0.000,B 0.000,C 90.000,E1 296.539} C_DIS
LIN {X 0.205,Y -538.047,Z 1102.439,A 0.000,B 0.000,C 90.000,E1 295.079} C_DIS
LIN {X 0.035,Y -538.551,Z 1102.430,A 0.000,B 0.000,C 90.000,E1 293.387} C_DIS
LIN {X 0.167,Y -538.910,Z 1102.421,A 0.000,B 0.000,C 90.000,E1 291.663} C_DIS
LIN {X -0.137,Y -539.056,Z 1102.414,A 0.000,B 0.000,C 90.000,E1 290.556} C_DIS
LIN {X 0.065,Y -538.999,Z 1102.408,A 0.000,B 0.000,C 90.000,E1 289.396} C_DIS
LIN {X -0.204,Y -538.775,Z 1102.400,A 0.000,B 0.000,C 90.000,E1 288.000} C_DIS
LIN {X 0.082,Y -538.408,Z 1102.390,A 0.000,B 0.000,C 90.000,E1 286.260} C_DIS
LIN {X 0.145,Y -537.866,Z 1102.383,A 0.000,B 0.000,C 90.000,E1 284.828} C_DIS
LIN {X 0.118,Y -537.088,Z 1102.373,A 0.000,B 0.000,C 90.000,E1 283.119} C_DIS
LIN {X 0.020,Y -536.101,Z 1102.362,A 0.000,B 0.000,C 90.000,E1 281.130} C_DIS
LIN {X -0.220,Y -535.362,Z 1102.354,A 0.000,B 0.000,C 90.000,E1 279.726} C_DIS
LIN {X -0.070,Y -534.546,Z 1102.344,A 0.000,B 0.000,C 90.000,E1 277.992} C_DIS
LIN {X 0.068,Y -533.704,Z 1102.335,A 0.000,B 0.000,C 90.000,E1 276.258} C_DIS
LIN {X 0.093,Y -533.044,Z 1102.327,A 0.000,B 0.000,C 90.000,E1 274.821} C_DIS
LIN {X 0.114,Y -532.103,Z 1102.316,A 0.000,B 0.000,C 90.000,E1 272.808} C_DIS
LIN {X 0.049,Y -531.179,Z 1102.305,A 0.000,B 0.000,C 90.000,E1 270.802} C_DIS
LIN {X -0.016,Y -530.460,Z 1102.297,A 0.000,B 0.000,C 90.000,E1 269.370} C_DIS
LIN {X -0.083,Y -529.738,Z 1102.289,A 0.000,B 0.000,C 90.000,E1 267.936} C_DIS
LIN {X -0.187,Y -528.668,Z 1102.279,A 0.000,B 0.000,C 90.000,E1 266.216} C_DIS
LIN {X -0.257,Y -527.774,Z 1102.271,A 0.000,B 0.000,C 90.000,E1 264.780} C_DIS
LIN {X 0.218,Y -526.912,Z 1102.265,A 0.000,B 0.000,C 90.000,E1 263.571} C_DIS
LIN {X 0.219,Y -525.772,Z 1102.258,A 0.000,B 0.000,C 90.000,E1 262.413} C_DIS
LIN {X 0.167,Y -523.679,Z 1102.247,A 0.000,B 0.000,C 90.000,E1 260.387} C_DIS
LIN {X 0.225,Y -522.284,Z 1102.239,A 0.000,B 0.000,C 90.000,E1 258.926} C_DIS
LIN {X -0.245,Y -520.293,Z 1102.227,A 0.000,B 0.000,C 90.000,E1 256.937} C_DIS
LIN {X -0.147,Y -518.638,Z 1102.218,A 0.000,B 0.000,C 90.000,E1 255.172} C_DIS
LIN {X 0.156,Y -516.505,Z 1102.206,A 0.000,B 0.000,C 90.000,E1 253.087} C_DIS
LIN {X 0.101,Y -514.623,Z 1102.196,A 0.000,B 0.000,C 90.000,E1 251.329} C_DIS
LIN {X -0.230,Y -513.341,Z 1102.190,A 0.000,B 0.000,C 90.000,E1 250.188} C_DIS
LIN {X -0.065,Y -510.951,Z 1102.178,A 0.000,B 0.000,C 90.000,E1 248.103} C_DIS
LIN {X -0.092,Y -509.543,Z 1102.172,A 0.000,B 0.000,C 90.000,E1 246.922} C_DIS
LIN {X -0.143,Y -507.802,Z 1102.165,A 0.000,B 0.000,C 90.000,E1 245.741} C_DIS
LIN {X 0.075,Y -505.544,Z 1102.157,A 0.000,B 0.000,C 90.000,E1 244.229} C_DIS
LIN {X 0.088,Y -502.587,Z 1102.147,A 0.000,B 0.000,C 90.000,E1 242.436} C_DIS
LIN {X 0.214,Y -500.133,Z 1102.139,A 0.000,B 0.000,C 90.000,E1 240.923} C_DIS
LIN {X -0.130,Y -497.618,Z 1102.130,A 0.000,B 0.000,C 90.000,E1 239.459} C_DIS
LIN {X 0.165,Y -494.960,Z 1102.122,A 0.000,B 0.000,C 90.000,E1 237.916} C_DIS
LIN {X 0.246,Y -491.751,Z 1102.112,A 0.000,B 0.000,C 90.000,E1 236.087} C_DIS
LIN {X 0.031,Y -489.548,Z 1102.105,A 0.000,B 0.000,C 90.000,E1 234.895} C_DIS
LIN {X 0.136,Y -486.045,Z 1102.095,A 0.000,B 0.000,C 90.000,E1 233.050} C_DIS
LIN {X 0.130,Y -483.665,Z 1102.088,A 0.000,B 0.000,C 90.000,E1 231.823} C_DIS
LIN {X 0.080,Y -481.165,Z 1102.081,A 0.000,B 0.000,C 90.000,E1 230.598} C_DIS
LIN {X 0.040,Y -478.061,Z 1102.073,A 0.000,B 0.000,C 90.000,E1 229.057} C_DIS
LIN {X -0.161,Y -473.811,Z 1102.061,A 0.000,B 0.000,C 90.000,E1 226.905} C_DIS
LIN {X 0.083,Y -470.426,Z 1102.050,A 0.000,B 0.000,C 90.000,E1 225.000} C_DIS
LIN {X -0.170,Y -467.576,Z 1102.041,A 0.000,B 0.000,C 90.000,E1 223.461} C_DIS
LIN {X -0.049,Y -464.090,Z 1102.031,A 0.000,B 0.000,C 90.000,E1 221.553} C_DIS
LIN {X -0.046,Y -461.280,Z 1102.022,A 0.000,B 0.000,C 90.000,E1 219.967} C_DIS
LIN {X -0.102,Y -458.584,Z 1102.013,A 0.000,B 0.000,C 90.000,E1 218.382} C_DIS
LIN {X -0.050,Y -455.429,Z 1102.003,A 0.000,B 0.000,C 90.000,E1 216.457} C_DIS
LIN {X 0.211,Y -452.938,Z 1101.994,A 0.000,B 0.000,C 90.000,E1 214.818} C_DIS
LIN {X -0.060,Y -449.455,Z 1101.981,A 0.000,B 0.000,C 90.000,E1 212.594} C_DIS
LIN {X -0.216,Y -446.552,Z 1101.970,A 0.000,B 0.000,C 90.000,E1 210.669} C_DIS
LIN {X -0.087,Y -442.620,Z 1101.954,A 0.000,B 0.000,C 90.000,E1 207.719} C_DIS
LIN {X -0.114,Y -439.488,Z 1101.938,A 0.000,B 0.000,C 90.000,E1 204.771} C_DIS
LIN {X -0.149,Y -438.548,Z 1101.928,A 0.000,B 0.000,C 90.000,E1 203.131} C_DIS
LIN {X -0.225,Y -438.503,Z 1101.923,A 0.000,B 0.000,C 90.000,E1 202.153} C_DIS
LIN {X -0.134,Y -439.003,Z 1101.917,A 0.000,B 0.000,C 90.000,E1 201.153} C_DIS
LIN {X -0.043,Y -439.643,Z 1101.914,A 0.000,B 0.000,C 90.000,E1 200.482} C_DIS
LIN {X 0.055,Y -440.711,Z 1101.910,A 0.000,B 0.000,C 90.000,E1 199.812} C_DIS
LIN {X -0.136,Y -442.894,Z 1101.905,A 0.000,B 0.000,C 90.000,E1 198.852} C_DIS
LIN {X -0.161,Y -445.628,Z 1101.899,A 0.000,B 0.000,C 90.000,E1 197.873} C_DIS
LIN {X 0.019,Y -450.671,Z 1101.891,A 0.000,B 0.000,C 90.000,E1 196.386} C_DIS
LIN {X -0.128,Y -462.932,Z 1101.874,A 0.000,B 0.000,C 90.000,E1 193.355} C_DIS
LIN {X 0.173,Y -471.167,Z 1101.864,A 0.000,B 0.000,C 90.000,E1 191.422} C_DIS
LIN {X 0.119,Y -479.831,Z 1101.853,A 0.000,B 0.000,C 90.000,E1 189.557} C_DIS
LIN {X -0.045,Y -485.620,Z 1101.846,A 0.000,B 0.000,C 90.000,E1 188.341} C_DIS
LIN {X -0.124,Y -491.295,Z 1101.840,A 0.000,B 0.000,C 90.000,E1 187.125} C_DIS
LIN {X 0.047,Y -497.571,Z 1101.832,A 0.000,B 0.000,C 90.000,E1 185.739} C_DIS
LIN {X 0.156,Y -505.066,Z 1101.823,A 0.000,B 0.000,C 90.000,E1 184.073} C_DIS
LIN {X 0.005,Y -511.184,Z 1101.815,A 0.000,B 0.000,C 90.000,E1 182.751} C_DIS
LIN {X -0.210,Y -520.013,Z 1101.805,A 0.000,B 0.000,C 90.000,E1 180.859} C_DIS
LIN {X 0.085,Y -526.838,Z 1101.797,A 0.000,B 0.000,C 90.000,E1 179.370} C_DIS
LIN {X -0.016,Y -534.975,Z 1101.787,A 0.000,B 0.000,C 90.000,E1 177.650} C_DIS
LIN {X 0.037,Y -541.702,Z 1101.779,A 0.000,B 0.000,C 90.000,E1 176.216} C_DIS
LIN {X -0.119,Y -546.312,Z 1101.774,A 0.000,B 0.000,C 90.000,E1 175.241} C_DIS
LIN {X -0.028,Y -553.560,Z 1101.765,A 0.000,B 0.000,C 90.000,E1 173.685} C_DIS
LIN {X 0.148,Y -559.490,Z 1101.758,A 0.000,B 0.000,C 90.000,E1 172.413} C_DIS
LIN {X -0.135,Y -565.344,Z 1101.751,A 0.000,B 0.000,C 90.000,E1 171.197} C_DIS
LIN {X -0.095,Y -570.452,Z 1101.745,A 0.000,B 0.000,C 90.000,E1 170.095} C_DIS
LIN {X 0.092,Y -577.252,Z 1101.737,A 0.000,B 0.000,C 90.000,E1 168.578} C_DIS
LIN {X 0.171,Y -582.578,Z 1101.730,A 0.000,B 0.000,C 90.000,E1 167.353} C_DIS
LIN {X -0.266,Y -586.003,Z 1101.725,A 0.000,B 0.000,C 90.000,E1 166.589} C_DIS
LIN {X -0.017,Y -591.444,Z 1101.718,A 0.000,B 0.000,C 90.000,E1 165.227} C_DIS
LIN {X -0.244,Y -596.531,Z 1101.711,A 0.000,B 0.000,C 90.000,E1 163.921} C_DIS
LIN {X 0.071,Y -600.306,Z 1101.705,A 0.000,B 0.000,C 90.000,E1 162.834} C_DIS
LIN {X 0.261,Y -603.891,Z 1101.699,A 0.000,B 0.000,C 90.000,E1 161.764} C_DIS
LIN {X 0.111,Y -607.179,Z 1101.693,A 0.000,B 0.000,C 90.000,E1 160.732} C_DIS
LIN {X -0.052,Y -611.103,Z 1101.686,A 0.000,B 0.000,C 90.000,E1 159.444} C_DIS
LIN {X -0.145,Y -614.797,Z 1101.679,A 0.000,B 0.000,C 90.000,E1 158.156} C_DIS
LIN {X 0.074,Y -617.644,Z 1101.673,A 0.000,B 0.000,C 90.000,E1 157.102} C_DIS
LIN {X 0.321,Y -621.093,Z 1101.666,A 0.000,B 0.000,C 90.000,E1 155.793} C_DIS
LIN {X 0.055,Y -624.390,Z 1101.659,A 0.000,B 0.000,C 90.000,E1 154.537} C_DIS
LIN {X 0.111,Y -627.577,Z 1101.651,A 0.000,B 0.000,C 90.000,E1 153.256} C_DIS
LIN {X 0.193,Y -629.895,Z 1101.646,A 0.000,B 0.000,C 90.000,E1 152.231} C_DIS
LIN {X 0.082,Y -632.737,Z 1101.639,A 0.000,B 0.000,C 90.000,E1 150.973} C_DIS
LIN {X -0.293,Y -635.505,Z 1101.632,A 0.000,B 0.000,C 90.000,E1 149.744} C_DIS
LIN {X 0.017,Y -638.139,Z 1101.625,A 0.000,B 0.000,C 90.000,E1 148.456} C_DIS
LIN {X 0.034,Y -640.634,Z 1101.618,A 0.000,B 0.000,C 90.000,E1 147.199} C_DIS
LIN {X -0.110,Y -643.039,Z 1101.611,A 0.000,B 0.000,C 90.000,E1 145.960} C_DIS
LIN {X 0.154,Y -645.325,Z 1101.604,A 0.000,B 0.000,C 90.000,E1 144.689} C_DIS
LIN {X -0.014,Y -648.021,Z 1101.596,A 0.000,B 0.000,C 90.000,E1 143.210} C_DIS
LIN {X -0.184,Y -650.263,Z 1101.589,A 0.000,B 0.000,C 90.000,E1 141.984} C_DIS
LIN {X 0.060,Y -653.498,Z 1101.579,A 0.000,B 0.000,C 90.000,E1 140.231} C_DIS
LIN {X 0.257,Y -657.316,Z 1101.568,A 0.000,B 0.000,C 90.000,E1 138.243} C_DIS
LIN {X 0.119,Y -660.298,Z 1101.560,A 0.000,B 0.000,C 90.000,E1 136.782} C_DIS
LIN {X -0.016,Y -665.087,Z 1101.548,A 0.000,B 0.000,C 90.000,E1 134.595} C_DIS
LIN {X -0.024,Y -669.750,Z 1101.537,A 0.000,B 0.000,C 90.000,E1 132.651} C_DIS
LIN {X 0.155,Y -673.991,Z 1101.528,A 0.000,B 0.000,C 90.000,E1 130.943} C_DIS
LIN {X -0.085,Y -677.540,Z 1101.520,A 0.000,B 0.000,C 90.000,E1 129.519} C_DIS
LIN {X 0.296,Y -681.877,Z 1101.510,A 0.000,B 0.000,C 90.000,E1 127.810} C_DIS
LIN {X -0.267,Y -684.952,Z 1101.504,A 0.000,B 0.000,C 90.000,E1 126.664} C_DIS
LIN {X 0.144,Y -687.318,Z 1101.498,A 0.000,B 0.000,C 90.000,E1 125.678} C_DIS
LIN {X 0.224,Y -690.254,Z 1101.492,A 0.000,B 0.000,C 90.000,E1 124.485} C_DIS
LIN {X 0.217,Y -694.271,Z 1101.483,A 0.000,B 0.000,C 90.000,E1 122.832} C_DIS
LIN {X -0.227,Y -696.544,Z 1101.477,A 0.000,B 0.000,C 90.000,E1 121.926} C_DIS
LIN {X -0.423,Y -698.617,Z 1101.472,A 0.000,B 0.000,C 90.000,E1 121.003} C_DIS
LIN {X 0.371,Y -700.425,Z 1101.467,A 0.000,B 0.000,C 90.000,E1 120.001} C_DIS
LIN {X 0.230,Y -701.959,Z 1101.462,A 0.000,B 0.000,C 90.000,E1 119.077} C_DIS
LIN {X 0.103,Y -703.256,Z 1101.457,A 0.000,B 0.000,C 90.000,E1 118.153} C_DIS
LIN {X -0.342,Y -704.217,Z 1101.451,A 0.000,B 0.000,C 90.000,E1 117.257} C_DIS
LIN {X -0.194,Y -705.294,Z 1101.444,A 0.000,B 0.000,C 90.000,E1 115.848} C_DIS
LIN {X -0.265,Y -705.651,Z 1101.440,A 0.000,B 0.000,C 90.000,E1 115.155} C_DIS
LIN {X 0.315,Y -705.639,Z 1101.437,A 0.000,B 0.000,C 90.000,E1 114.643} C_DIS
LIN {X -0.041,Y -705.097,Z 1101.435,A 0.000,B 0.000,C 90.000,E1 114.207} C_DIS
LIN {X 0.247,Y -704.726,Z 1101.433,A 0.000,B 0.000,C 90.000,E1 113.951} C_DIS
LIN {X -0.113,Y -702.967,Z 1101.431,A 0.000,B 0.000,C 90.000,E1 113.515} C_DIS
LIN {X 0.167,Y -701.879,Z 1101.429,A 0.000,B 0.000,C 90.000,E1 113.259} C_DIS
LIN {X -0.116,Y -698.000,Z 1101.427,A 0.000,B 0.000,C 90.000,E1 112.823} C_DIS
LIN {X 0.014,Y -696.880,Z 1101.426,A 0.000,B 0.000,C 90.000,E1 112.695} C_DIS
LIN {X -0.124,Y -695.202,Z 1101.426,A 0.000,B 0.000,C 90.000,E1 112.589} C_DIS
LIN {X -0.181,Y -687.345,Z 1101.424,A 0.000,B 0.000,C 90.000,E1 112.259} C_DIS
LIN {X 0.279,Y -685.423,Z 1101.423,A 0.000,B 0.000,C 90.000,E1 112.153} C_DIS
LIN {X -0.126,Y -683.457,Z 1101.423,A 0.000,B 0.000,C 90.000,E1 112.153} C_DIS
LIN {X -0.267,Y -676.203,Z 1101.423,A 0.000,B 0.000,C 90.000,E1 112.078} C_DIS
LIN {X 0.273,Y -604.207,Z 1101.423,A 0.000,B 0.000,C 90.000,E1 112.025} C_DIS
LIN {X 0.111,Y -600.556,Z 1101.422,A 0.000,B 0.000,C 90.000,E1 111.844} C_DIS
LIN {X 0.047,Y -596.043,Z 1101.420,A 0.000,B 0.000,C 90.000,E1 111.535} C_DIS
LIN {X 0.208,Y -578.921,Z 1101.412,A 0.000,B 0.000,C 90.000,E1 110.066} C_DIS
LIN {X -0.284,Y -574.726,Z 1101.410,A 0.000,B 0.000,C 90.000,E1 109.758} C_DIS
LIN {X 0.050,Y -568.626,Z 1101.407,A 0.000,B 0.000,C 90.000,E1 109.268} C_DIS
LIN {X -0.212,Y -560.314,Z 1101.404,A 0.000,B 0.000,C 90.000,E1 108.779} C_DIS
LIN {X 0.211,Y -553.902,Z 1101.402,A 0.000,B 0.000,C 90.000,E1 108.362} C_DIS
LIN {X 0.195,Y -549.781,Z 1101.401,A 0.000,B 0.000,C 90.000,E1 108.055} C_DIS
LIN {X 0.129,Y -548.459,Z 1101.399,A 0.000,B 0.000,C 90.000,E1 107.873} C_DIS
LIN {X 0.088,Y -548.434,Z 1101.399,A 0.000,B 0.000,C 90.000,E1 107.873} C_DIS
LIN {X 0.176,Y -548.134,Z 1101.398,A 0.000,B 0.000,C 90.000,E1 107.583} C_DIS
LIN {X 0.215,Y -548.445,Z 1101.393,A 0.000,B 0.000,C 90.000,E1 106.677} C_DIS
LIN {X 0.143,Y -549.772,Z 1101.382,A 0.000,B 0.000,C 90.000,E1 104.717} C_DIS
LIN {X 0.202,Y -551.801,Z 1101.368,A 0.000,B 0.000,C 90.000,E1 102.187} C_DIS
LIN {X -0.162,Y -553.393,Z 1101.359,A 0.000,B 0.000,C 90.000,E1 100.546} C_DIS
LIN {X 0.069,Y -555.397,Z 1101.348,A 0.000,B 0.000,C 90.000,E1 98.568} C_DIS
LIN {X 0.002,Y -556.820,Z 1101.340,A 0.000,B 0.000,C 90.000,E1 97.182} C_DIS
LIN {X -0.039,Y -558.288,Z 1101.332,A 0.000,B 0.000,C 90.000,E1 95.796} C_DIS
LIN {X 0.238,Y -559.102,Z 1101.328,A 0.000,B 0.000,C 90.000,E1 94.935} C_DIS
LIN {X 0.095,Y -560.011,Z 1101.321,A 0.000,B 0.000,C 90.000,E1 93.841} C_DIS
LIN {X 0.012,Y -560.882,Z 1101.314,A 0.000,B 0.000,C 90.000,E1 92.465} C_DIS
LIN {X -0.246,Y -561.373,Z 1101.309,A 0.000,B 0.000,C 90.000,E1 91.661} C_DIS
LIN {X 0.144,Y -561.956,Z 1101.303,A 0.000,B 0.000,C 90.000,E1 90.516} C_DIS
LIN {X 0.187,Y -562.761,Z 1101.294,A 0.000,B 0.000,C 90.000,E1 88.854} C_DIS
LIN {X 0.154,Y -563.390,Z 1101.286,A 0.000,B 0.000,C 90.000,E1 87.478} C_DIS
LIN {X 0.130,Y -563.976,Z 1101.278,A 0.000,B 0.000,C 90.000,E1 86.102} C_DIS
LIN {X 0.151,Y -564.529,Z 1101.271,A 0.000,B 0.000,C 90.000,E1 84.723} C_DIS
LIN {X 0.242,Y -565.049,Z 1101.263,A 0.000,B 0.000,C 90.000,E1 83.337} C_DIS
LIN {X -0.214,Y -565.529,Z 1101.255,A 0.000,B 0.000,C 90.000,E1 82.008} C_DIS
LIN {X 0.060,Y -566.072,Z 1101.246,A 0.000,B 0.000,C 90.000,E1 80.330} C_DIS
LIN {X 0.189,Y -566.568,Z 1101.240,A 0.000,B 0.000,C 90.000,E1 79.218} C_DIS
LIN {X 0.012,Y -567.356,Z 1101.231,A 0.000,B 0.000,C 90.000,E1 77.589} C_DIS
LIN {X 0.288,Y -567.914,Z 1101.225,A 0.000,B 0.000,C 90.000,E1 76.464} C_DIS
LIN {X 0.185,Y -569.164,Z 1101.213,A 0.000,B 0.000,C 90.000,E1 74.283} C_DIS
LIN {X -0.131,Y -570.789,Z 1101.201,A 0.000,B 0.000,C 90.000,E1 72.127} C_DIS
LIN {X 0.145,Y -572.336,Z 1101.190,A 0.000,B 0.000,C 90.000,E1 70.188} C_DIS
LIN {X -0.240,Y -573.830,Z 1101.181,A 0.000,B 0.000,C 90.000,E1 68.592} C_DIS
LIN {X -0.007,Y -575.475,Z 1101.170,A 0.000,B 0.000,C 90.000,E1 66.666} C_DIS
LIN {X -0.118,Y -576.833,Z 1101.161,A 0.000,B 0.000,C 90.000,E1 65.049} C_DIS
LIN {X 0.139,Y -578.175,Z 1101.151,A 0.000,B 0.000,C 90.000,E1 63.127} C_DIS
LIN {X 0.201,Y -579.125,Z 1101.143,A 0.000,B 0.000,C 90.000,E1 61.769} C_DIS
LIN {X -0.087,Y -580.096,Z 1101.134,A 0.000,B 0.000,C 90.000,E1 60.177} C_DIS
LIN {X -0.009,Y -580.850,Z 1101.127,A 0.000,B 0.000,C 90.000,E1 58.820} C_DIS
LIN {X 0.178,Y -581.597,Z 1101.119,A 0.000,B 0.000,C 90.000,E1 57.454} C_DIS
LIN {X -0.080,Y -582.590,Z 1101.109,A 0.000,B 0.000,C 90.000,E1 55.595} C_DIS
LIN {X -0.165,Y -583.259,Z 1101.100,A 0.000,B 0.000,C 90.000,E1 53.989} C_DIS
LIN {X -0.261,Y -583.664,Z 1101.094,A 0.000,B 0.000,C 90.000,E1 52.924} C_DIS
LIN {X 0.004,Y -583.967,Z 1101.088,A 0.000,B 0.000,C 90.000,E1 51.823} C_DIS
LIN {X -0.089,Y -584.119,Z 1101.085,A 0.000,B 0.000,C 90.000,E1 51.295} C_DIS
LIN {X 0.188,Y -584.082,Z 1101.079,A 0.000,B 0.000,C 90.000,E1 50.194} C_DIS
LIN {X 0.189,Y -583.895,Z 1101.072,A 0.000,B 0.000,C 90.000,E1 48.852} C_DIS
LIN {X -0.259,Y -583.527,Z 1101.064,A 0.000,B 0.000,C 90.000,E1 47.553} C_DIS
LIN {X -0.058,Y -583.128,Z 1101.058,A 0.000,B 0.000,C 90.000,E1 46.458} C_DIS
LIN {X 0.279,Y -582.413,Z 1101.051,A 0.000,B 0.000,C 90.000,E1 45.081} C_DIS
LIN {X 0.045,Y -581.675,Z 1101.045,A 0.000,B 0.000,C 90.000,E1 44.028} C_DIS
LIN {X 0.221,Y -580.569,Z 1101.039,A 0.000,B 0.000,C 90.000,E1 42.933} C_DIS
LIN {X -0.052,Y -579.322,Z 1101.033,A 0.000,B 0.000,C 90.000,E1 41.881} C_DIS
LIN {X -0.020,Y -578.235,Z 1101.028,A 0.000,B 0.000,C 90.000,E1 41.067} C_DIS
LIN {X -0.281,Y -576.578,Z 1101.022,A 0.000,B 0.000,C 90.000,E1 40.011} C_DIS
LIN {X -0.121,Y -574.713,Z 1101.016,A 0.000,B 0.000,C 90.000,E1 38.910} C_DIS
LIN {X -0.128,Y -572.997,Z 1101.012,A 0.000,B 0.000,C 90.000,E1 38.096} C_DIS
LIN {X -0.160,Y -571.166,Z 1101.007,A 0.000,B 0.000,C 90.000,E1 37.282} C_DIS
LIN {X 0.109,Y -569.794,Z 1101.004,A 0.000,B 0.000,C 90.000,E1 36.710} C_DIS
LIN {X 0.159,Y -567.399,Z 1101.000,A 0.000,B 0.000,C 90.000,E1 35.884} C_DIS
LIN {X -0.060,Y -565.654,Z 1100.996,A 0.000,B 0.000,C 90.000,E1 35.358} C_DIS
LIN {X 0.054,Y -561.580,Z 1100.990,A 0.000,B 0.000,C 90.000,E1 34.246} C_DIS
LIN {X 0.021,Y -558.056,Z 1100.986,A 0.000,B 0.000,C 90.000,E1 33.420} C_DIS
LIN {X -0.049,Y -554.232,Z 1100.981,A 0.000,B 0.000,C 90.000,E1 32.594} C_DIS
LIN {X 0.009,Y -550.092,Z 1100.976,A 0.000,B 0.000,C 90.000,E1 31.750} C_DIS
LIN {X 0.343,Y -544.068,Z 1100.970,A 0.000,B 0.000,C 90.000,E1 30.590} C_DIS
LIN {X 0.034,Y -537.398,Z 1100.964,A 0.000,B 0.000,C 90.000,E1 29.489} C_DIS
LIN {X -0.253,Y -533.720,Z 1100.961,A 0.000,B 0.000,C 90.000,E1 28.949} C_DIS
LIN {X 0.072,Y -527.807,Z 1100.956,A 0.000,B 0.000,C 90.000,E1 28.052} C_DIS
LIN {X 0.022,Y -522.327,Z 1100.952,A 0.000,B 0.000,C 90.000,E1 27.334} C_DIS
LIN {X 0.086,Y -517.630,Z 1100.949,A 0.000,B 0.000,C 90.000,E1 26.744} C_DIS
LIN {X -0.048,Y -511.260,Z 1100.945,A 0.000,B 0.000,C 90.000,E1 26.027} C_DIS
LIN {X 0.191,Y -503.448,Z 1100.940,A 0.000,B 0.000,C 90.000,E1 25.155} C_DIS
LIN {X 0.001,Y -496.548,Z 1100.936,A 0.000,B 0.000,C 90.000,E1 24.463} C_DIS
LIN {X -0.007,Y -489.604,Z 1100.932,A 0.000,B 0.000,C 90.000,E1 23.770} C_DIS
LIN {X 0.093,Y -482.425,Z 1100.928,A 0.000,B 0.000,C 90.000,E1 23.078} C_DIS
LIN {X -0.156,Y -476.849,Z 1100.925,A 0.000,B 0.000,C 90.000,E1 22.589} C_DIS
LIN {X 0.054,Y -465.088,Z 1100.920,A 0.000,B 0.000,C 90.000,E1 21.535} C_DIS
LIN {X -0.075,Y -450.278,Z 1100.912,A 0.000,B 0.000,C 90.000,E1 20.248} C_DIS
LIN {X -0.038,Y -431.599,Z 1100.903,A 0.000,B 0.000,C 90.000,E1 18.489} C_DIS
LIN {X -0.152,Y -420.320,Z 1100.896,A 0.000,B 0.000,C 90.000,E1 17.330} C_DIS
LIN {X 0.020,Y -410.698,Z 1100.890,A 0.000,B 0.000,C 90.000,E1 16.205} C_DIS
LIN {X -0.181,Y -402.909,Z 1100.885,A 0.000,B 0.000,C 90.000,E1 15.245} C_DIS
LIN {X -0.044,Y -397.258,Z 1100.880,A 0.000,B 0.000,C 90.000,E1 14.411} C_DIS
LIN {X -0.045,Y -395.167,Z 1100.878,A 0.000,B 0.000,C 90.000,E1 14.008} C_DIS
LIN {X 0.144,Y -392.768,Z 1100.874,A 0.000,B 0.000,C 90.000,E1 13.300} C_DIS
LIN {X -0.022,Y -392.102,Z 1100.871,A 0.000,B 0.000,C 90.000,E1 12.703} C_DIS
LIN {X -0.117,Y -392.350,Z 1100.867,A 0.000,B 0.000,C 90.000,E1 12.007} C_DIS
LIN {X -0.191,Y -393.485,Z 1100.862,A 0.000,B 0.000,C 90.000,E1 11.130} C_DIS
LIN {X 0.001,Y -398.991,Z 1100.846,A 0.000,B 0.000,C 90.000,E1 8.276} C_DIS
LIN {X -0.123,Y -402.419,Z 1100.838,A 0.000,B 0.000,C 90.000,E1 6.891} C_DIS
LIN {X 0.170,Y -405.724,Z 1100.830,A 0.000,B 0.000,C 90.000,E1 5.454} C_DIS
LIN {X 0.170,Y -406.683,Z 1100.828,A 0.000,B 0.000,C 90.000,E1 5.106} C_DIS
LIN {X 0.172,Y -408.078,Z 1100.827,A 0.000,B 0.000,C 90.000,E1 4.759} C_DIS
LIN {X -0.124,Y -409.586,Z 1100.825,A 0.000,B 0.000,C 90.000,E1 4.473} C_DIS
LIN {X -0.145,Y -411.709,Z 1100.823,A 0.000,B 0.000,C 90.000,E1 4.131} C_DIS
LIN {X -0.080,Y -416.240,Z 1100.820,A 0.000,B 0.000,C 90.000,E1 3.669} C_DIS
LIN {X 0.142,Y -423.704,Z 1100.817,A 0.000,B 0.000,C 90.000,E1 3.094} C_DIS
LIN {X 0.214,Y -444.877,Z 1100.809,A 0.000,B 0.000,C 90.000,E1 1.661} C_DIS
LIN {X 0.076,Y -465.705,Z 1100.802,A 0.000,B 0.000,C 90.000,E1 0.344} C_DIS
LIN {X -0.112,Y -477.878,Z 1100.798,A 0.000,B 0.000,C 90.000,E1 359.599} C_DIS
LIN {X -0.012,Y -489.130,Z 1100.794,A 0.000,B 0.000,C 90.000,E1 358.854} C_DIS
LIN {X -0.071,Y -498.339,Z 1100.790,A 0.000,B 0.000,C 90.000,E1 358.224} C_DIS
LIN {X 0.031,Y -502.980,Z 1100.788,A 0.000,B 0.000,C 90.000,E1 357.879} C_DIS
LIN {X 0.110,Y -510.229,Z 1100.785,A 0.000,B 0.000,C 90.000,E1 357.306} C_DIS
LIN {X -0.072,Y -516.115,Z 1100.782,A 0.000,B 0.000,C 90.000,E1 356.846} C_DIS
LIN {X 0.065,Y -522.945,Z 1100.779,A 0.000,B 0.000,C 90.000,E1 356.216} C_DIS
LIN {X -0.152,Y -529.596,Z 1100.775,A 0.000,B 0.000,C 90.000,E1 355.584} C_DIS
LIN {X 0.108,Y -534.676,Z 1100.772,A 0.000,B 0.000,C 90.000,E1 355.008} C_DIS
LIN {X 0.000,Y -540.536,Z 1100.768,A 0.000,B 0.000,C 90.000,E1 354.318} C_DIS
LIN {X -0.193,Y -545.838,Z 1100.765,A 0.000,B 0.000,C 90.000,E1 353.628} C_DIS
LIN {X -0.084,Y -549.800,Z 1100.761,A 0.000,B 0.000,C 90.000,E1 353.053} C_DIS
LIN {X 0.123,Y -553.414,Z 1100.758,A 0.000,B 0.000,C 90.000,E1 352.470} C_DIS
LIN {X 0.034,Y -557.372,Z 1100.754,A 0.000,B 0.000,C 90.000,E1 351.781} C_DIS
LIN {X 0.057,Y -560.910,Z 1100.750,A 0.000,B 0.000,C 90.000,E1 351.084} C_DIS
LIN {X 0.114,Y -564.150,Z 1100.747,A 0.000,B 0.000,C 90.000,E1 350.387} C_DIS
LIN {X 0.055,Y -567.710,Z 1100.742,A 0.000,B 0.000,C 90.000,E1 349.567} C_DIS
LIN {X -0.074,Y -571.008,Z 1100.738,A 0.000,B 0.000,C 90.000,E1 348.757} C_DIS
LIN {X 0.135,Y -575.031,Z 1100.731,A 0.000,B 0.000,C 90.000,E1 347.645} C_DIS
LIN {X 0.051,Y -579.586,Z 1100.724,A 0.000,B 0.000,C 90.000,E1 346.297} C_DIS
LIN {X 0.000,Y -584.672,Z 1100.715,A 0.000,B 0.000,C 90.000,E1 344.685} C_DIS
LIN {X -0.017,Y -587.847,Z 1100.709,A 0.000,B 0.000,C 90.000,E1 343.614} C_DIS
LIN {X 0.003,Y -590.961,Z 1100.703,A 0.000,B 0.000,C 90.000,E1 342.543} C_DIS
LIN {X 0.242,Y -593.949,Z 1100.697,A 0.000,B 0.000,C 90.000,E1 341.456} C_DIS
LIN {X 0.069,Y -596.037,Z 1100.693,A 0.000,B 0.000,C 90.000,E1 340.678} C_DIS
LIN {X -0.288,Y -599.074,Z 1100.685,A 0.000,B 0.000,C 90.000,E1 339.390} C_DIS
LIN {X 0.268,Y -601.303,Z 1100.680,A 0.000,B 0.000,C 90.000,E1 338.284} C_DIS
LIN {X 0.229,Y -603.634,Z 1100.672,A 0.000,B 0.000,C 90.000,E1 336.975} C_DIS
LIN {X 0.290,Y -605.090,Z 1100.666,A 0.000,B 0.000,C 90.000,E1 335.921} C_DIS
LIN {X -0.135,Y -606.191,Z 1100.662,A 0.000,B 0.000,C 90.000,E1 335.177} C_DIS
LIN {X 0.148,Y -607.528,Z 1100.655,A 0.000,B 0.000,C 90.000,E1 333.845} C_DIS
LIN {X 0.051,Y -608.016,Z 1100.652,A 0.000,B 0.000,C 90.000,E1 333.332} C_DIS
LIN {X 0.144,Y -608.588,Z 1100.646,A 0.000,B 0.000,C 90.000,E1 332.281} C_DIS
LIN {X -0.036,Y -608.927,Z 1100.640,A 0.000,B 0.000,C 90.000,E1 331.257} C_DIS
LIN {X 0.123,Y -608.933,Z 1100.636,A 0.000,B 0.000,C 90.000,E1 330.461} C_DIS
LIN {X 0.233,Y -608.381,Z 1100.630,A 0.000,B 0.000,C 90.000,E1 329.410} C_DIS
LIN {X -0.191,Y -607.174,Z 1100.624,A 0.000,B 0.000,C 90.000,E1 328.408} C_DIS
LIN {X 0.203,Y -605.562,Z 1100.619,A 0.000,B 0.000,C 90.000,E1 327.327} C_DIS
LIN {X 0.142,Y -603.931,Z 1100.614,A 0.000,B 0.000,C 90.000,E1 326.548} C_DIS
LIN {X -0.265,Y -602.186,Z 1100.610,A 0.000,B 0.000,C 90.000,E1 325.801} C_DIS
LIN {X -0.104,Y -600.879,Z 1100.607,A 0.000,B 0.000,C 90.000,E1 325.261} C_DIS
LIN {X 0.143,Y -600.314,Z 1100.606,A 0.000,B 0.000,C 90.000,E1 324.975} C_DIS
LIN {X 0.038,Y -598.354,Z 1100.601,A 0.000,B 0.000,C 90.000,E1 324.196} C_DIS
LIN {X -0.099,Y -594.939,Z 1100.594,A 0.000,B 0.000,C 90.000,E1 322.889} C_DIS
LIN {X 0.181,Y -591.664,Z 1100.586,A 0.000,B 0.000,C 90.000,E1 321.537} C_DIS
LIN {X -0.075,Y -588.178,Z 1100.579,A 0.000,B 0.000,C 90.000,E1 320.231} C_DIS
LIN {X 0.360,Y -584.664,Z 1100.572,A 0.000,B 0.000,C 90.000,E1 318.852} C_DIS
LIN {X 0.276,Y -583.186,Z 1100.569,A 0.000,B 0.000,C 90.000,E1 318.324} C_DIS
LIN {X -0.086,Y -580.541,Z 1100.564,A 0.000,B 0.000,C 90.000,E1 317.553} C_DIS
LIN {X -0.078,Y -577.514,Z 1100.560,A 0.000,B 0.000,C 90.000,E1 316.743} C_DIS
LIN {X -0.214,Y -575.339,Z 1100.557,A 0.000,B 0.000,C 90.000,E1 316.215} C_DIS
LIN {X 0.293,Y -572.275,Z 1100.553,A 0.000,B 0.000,C 90.000,E1 315.486} C_DIS
LIN {X 0.211,Y -568.054,Z 1100.548,A 0.000,B 0.000,C 90.000,E1 314.676} C_DIS
LIN {X 0.155,Y -566.051,Z 1100.546,A 0.000,B 0.000,C 90.000,E1 314.271} C_DIS
LIN {X -0.145,Y -561.051,Z 1100.541,A 0.000,B 0.000,C 90.000,E1 313.338} C_DIS
LIN {X 0.218,Y -557.183,Z 1100.537,A 0.000,B 0.000,C 90.000,E1 312.609} C_DIS
LIN {X 0.164,Y -553.094,Z 1100.533,A 0.000,B 0.000,C 90.000,E1 311.919} C_DIS
LIN {X 0.076,Y -548.886,Z 1100.529,A 0.000,B 0.000,C 90.000,E1 311.229} C_DIS
LIN {X -0.050,Y -544.833,Z 1100.525,A 0.000,B 0.000,C 90.000,E1 310.539} C_DIS
LIN {X -0.015,Y -543.478,Z 1100.524,A 0.000,B 0.000,C 90.000,E1 310.253} C_DIS
LIN {X 0.017,Y -541.916,Z 1100.522,A 0.000,B 0.000,C 90.000,E1 309.967} C_DIS
LIN {X -0.027,Y -540.806,Z 1100.521,A 0.000,B 0.000,C 90.000,E1 309.688} C_DIS
LIN {X -0.188,Y -540.127,Z 1100.520,A 0.000,B 0.000,C 90.000,E1 309.564} C_DIS
LIN {X -0.168,Y -539.148,Z 1100.518,A 0.000,B 0.000,C 90.000,E1 309.277} C_DIS
LIN {X 0.203,Y -537.646,Z 1100.515,A 0.000,B 0.000,C 90.000,E1 308.669} C_DIS
LIN {X 0.239,Y -535.424,Z 1100.509,A 0.000,B 0.000,C 90.000,E1 307.523} C_DIS
LIN {X 0.247,Y -534.916,Z 1100.505,A 0.000,B 0.000,C 90.000,E1 306.950} C_DIS
LIN {X -0.128,Y -534.871,Z 1100.504,A 0.000,B 0.000,C 90.000,E1 306.710} C_DIS
LIN {X -0.287,Y -534.350,Z 1100.502,A 0.000,B 0.000,C 90.000,E1 306.297} C_DIS
LIN {X -0.052,Y -534.362,Z 1100.500,A 0.000,B 0.000,C 90.000,E1 305.964} C_DIS
LIN {X -0.052,Y -534.025,Z 1100.497,A 0.000,B 0.000,C 90.000,E1 305.391} C_DIS
LIN {X -0.054,Y -534.054,Z 1100.495,A 0.000,B 0.000,C 90.000,E1 305.105} C_DIS
LIN {X -0.058,Y -533.920,Z 1100.493,A 0.000,B 0.000,C 90.000,E1 304.818} C_DIS
LIN {X -0.069,Y -534.017,Z 1100.490,A 0.000,B 0.000,C 90.000,E1 304.246} C_DIS
LIN {X 0.367,Y -533.921,Z 1100.489,A 0.000,B 0.000,C 90.000,E1 303.913} C_DIS
LIN {X 0.059,Y -534.088,Z 1100.485,A 0.000,B 0.000,C 90.000,E1 303.372} C_DIS
LIN {X -0.120,Y -534.679,Z 1100.476,A 0.000,B 0.000,C 90.000,E1 301.671} C_DIS
LIN {X 0.168,Y -535.796,Z 1100.466,A 0.000,B 0.000,C 90.000,E1 299.922} C_DIS
LIN {X 0.221,Y -536.641,Z 1100.458,A 0.000,B 0.000,C 90.000,E1 298.487} C_DIS
LIN {X 0.218,Y -537.636,Z 1100.447,A 0.000,B 0.000,C 90.000,E1 296.488} C_DIS
LIN {X 0.055,Y -538.245,Z 1100.439,A 0.000,B 0.000,C 90.000,E1 295.079} C_DIS
LIN {X 0.163,Y -538.702,Z 1100.432,A 0.000,B 0.000,C 90.000,E1 293.643} C_DIS
LIN {X 0.027,Y -539.172,Z 1100.420,A 0.000,B 0.000,C 90.000,E1 291.663} C_DIS
LIN {X -0.084,Y -539.329,Z 1100.414,A 0.000,B 0.000,C 90.000,E1 290.536} C_DIS
LIN {X -0.068,Y -539.301,Z 1100.408,A 0.000,B 0.000,C 90.000,E1 289.396} C_DIS
LIN {X 0.181,Y -539.076,Z 1100.400,A 0.000,B 0.000,C 90.000,E1 287.946} C_DIS
LIN {X -0.038,Y -538.728,Z 1100.390,A 0.000,B 0.000,C 90.000,E1 286.260} C_DIS
LIN {X 0.030,Y -538.175,Z 1100.382,A 0.000,B 0.000,C 90.000,E1 284.828} C_DIS
LIN {X 0.010,Y -537.429,Z 1100.373,A 0.000,B 0.000,C 90.000,E1 283.119} C_DIS
LIN {X -0.079,Y -536.432,Z 1100.362,A 0.000,B 0.000,C 90.000,E1 281.130} C_DIS
LIN {X 0.158,Y -535.839,Z 1100.355,A 0.000,B 0.000,C 90.000,E1 279.962} C_DIS
LIN {X -0.131,Y -535.026,Z 1100.346,A 0.000,B 0.000,C 90.000,E1 278.276} C_DIS
LIN {X -0.010,Y -534.052,Z 1100.335,A 0.000,B 0.000,C 90.000,E1 276.258} C_DIS
LIN {X 0.021,Y -533.376,Z 1100.327,A 0.000,B 0.000,C 90.000,E1 274.821} C_DIS
LIN {X 0.050,Y -532.432,Z 1100.316,A 0.000,B 0.000,C 90.000,E1 272.808} C_DIS
LIN {X -0.017,Y -531.401,Z 1100.303,A 0.000,B 0.000,C 90.000,E1 270.516} C_DIS
LIN {X -0.094,Y -530.504,Z 1100.293,A 0.000,B 0.000,C 90.000,E1 268.797} C_DIS
LIN {X -0.162,Y -529.706,Z 1100.285,A 0.000,B 0.000,C 90.000,E1 267.364} C_DIS
LIN {X -0.239,Y -528.614,Z 1100.276,A 0.000,B 0.000,C 90.000,E1 265.641} C_DIS
LIN {X 0.217,Y -527.664,Z 1100.268,A 0.000,B 0.000,C 90.000,E1 264.147} C_DIS
LIN {X 0.163,Y -526.683,Z 1100.261,A 0.000,B 0.000,C 90.000,E1 262.996} C_DIS
LIN {X 0.126,Y -524.542,Z 1100.250,A 0.000,B 0.000,C 90.000,E1 260.971} C_DIS
LIN {X 0.205,Y -522.831,Z 1100.240,A 0.000,B 0.000,C 90.000,E1 259.218} C_DIS
LIN {X 0.258,Y -520.828,Z 1100.229,A 0.000,B 0.000,C 90.000,E1 257.173} C_DIS
LIN {X -0.143,Y -518.922,Z 1100.218,A 0.000,B 0.000,C 90.000,E1 255.172} C_DIS
LIN {X 0.190,Y -517.120,Z 1100.208,A 0.000,B 0.000,C 90.000,E1 253.378} C_DIS
LIN {X 0.118,Y -514.900,Z 1100.196,A 0.000,B 0.000,C 90.000,E1 251.329} C_DIS
LIN {X -0.208,Y -513.597,Z 1100.190,A 0.000,B 0.000,C 90.000,E1 250.188} C_DIS
LIN {X -0.036,Y -511.252,Z 1100.178,A 0.000,B 0.000,C 90.000,E1 248.103} C_DIS
LIN {X -0.061,Y -509.820,Z 1100.172,A 0.000,B 0.000,C 90.000,E1 246.922} C_DIS
LIN {X -0.107,Y -508.081,Z 1100.165,A 0.000,B 0.000,C 90.000,E1 245.741} C_DIS
LIN {X 0.116,Y -505.801,Z 1100.157,A 0.000,B 0.000,C 90.000,E1 244.229} C_DIS
LIN {X 0.134,Y -502.825,Z 1100.147,A 0.000,B 0.000,C 90.000,E1 242.436} C_DIS
LIN {X 0.264,Y -500.368,Z 1100.139,A 0.000,B 0.000,C 90.000,E1 240.923} C_DIS
LIN {X -0.075,Y -497.851,Z 1100.130,A 0.000,B 0.000,C 90.000,E1 239.459} C_DIS
LIN {X -0.186,Y -494.641,Z 1100.120,A 0.000,B 0.000,C 90.000,E1 237.661} C_DIS
LIN {X 0.157,Y -491.429,Z 1100.110,A 0.000,B 0.000,C 90.000,E1 235.801} C_DIS
LIN {X -0.060,Y -489.166,Z 1100.103,A 0.000,B 0.000,C 90.000,E1 234.609} C_DIS
LIN {X 0.038,Y -485.593,Z 1100.093,A 0.000,B 0.000,C 90.000,E1 232.763} C_DIS
LIN {X 0.022,Y -483.202,Z 1100.086,A 0.000,B 0.000,C 90.000,E1 231.537} C_DIS
LIN {X 0.153,Y -481.287,Z 1100.081,A 0.000,B 0.000,C 90.000,E1 230.598} C_DIS
LIN {X -0.198,Y -478.192,Z 1100.073,A 0.000,B 0.000,C 90.000,E1 229.094} C_DIS
LIN {X -0.083,Y -473.925,Z 1100.061,A 0.000,B 0.000,C 90.000,E1 226.905} C_DIS
LIN {X 0.162,Y -470.535,Z 1100.050,A 0.000,B 0.000,C 90.000,E1 225.000} C_DIS
LIN {X -0.089,Y -467.682,Z 1100.041,A 0.000,B 0.000,C 90.000,E1 223.461} C_DIS
LIN {X 0.033,Y -464.150,Z 1100.031,A 0.000,B 0.000,C 90.000,E1 221.553} C_DIS
LIN {X -0.061,Y -461.881,Z 1100.024,A 0.000,B 0.000,C 90.000,E1 220.297} C_DIS
LIN {X -0.046,Y -459.098,Z 1100.015,A 0.000,B 0.000,C 90.000,E1 218.705} C_DIS
LIN {X 0.122,Y -454.341,Z 1099.999,A 0.000,B 0.000,C 90.000,E1 215.804} C_DIS
LIN {X -0.190,Y -451.228,Z 1099.988,A 0.000,B 0.000,C 90.000,E1 213.913} C_DIS
LIN {X 0.093,Y -448.759,Z 1099.979,A 0.000,B 0.000,C 90.000,E1 212.260} C_DIS
LIN {X -0.220,Y -446.762,Z 1099.972,A 0.000,B 0.000,C 90.000,E1 211.003} C_DIS
LIN {X 0.072,Y -443.061,Z 1099.958,A 0.000,B 0.000,C 90.000,E1 208.359} C_DIS
LIN {X -0.215,Y -440.182,Z 1099.945,A 0.000,B 0.000,C 90.000,E1 206.104} C_DIS
LIN {X -0.076,Y -438.812,Z 1099.938,A 0.000,B 0.000,C 90.000,E1 204.771} C_DIS
LIN {X 0.116,Y -437.578,Z 1099.927,A 0.000,B 0.000,C 90.000,E1 202.770} C_DIS
LIN {X 0.197,Y -437.515,Z 1099.921,A 0.000,B 0.000,C 90.000,E1 201.770} C_DIS
LIN {X 0.114,Y -438.045,Z 1099.916,A 0.000,B 0.000,C 90.000,E1 200.791} C_DIS
LIN {X 0.199,Y -438.750,Z 1099.912,A 0.000,B 0.000,C 90.000,E1 200.120} C_DIS
LIN {X -0.123,Y -439.858,Z 1099.908,A 0.000,B 0.000,C 90.000,E1 199.504} C_DIS
LIN {X 0.094,Y -442.152,Z 1099.903,A 0.000,B 0.000,C 90.000,E1 198.489} C_DIS
LIN {X 0.060,Y -445.035,Z 1099.897,A 0.000,B 0.000,C 90.000,E1 197.511} C_DIS
LIN {X 0.086,Y -449.695,Z 1099.890,A 0.000,B 0.000,C 90.000,E1 196.205} C_DIS
LIN {X -0.048,Y -460.117,Z 1099.876,A 0.000,B 0.000,C 90.000,E1 193.647} C_DIS
LIN {X 0.186,Y -468.436,Z 1099.865,A 0.000,B 0.000,C 90.000,E1 191.715} C_DIS
LIN {X -0.204,Y -477.885,Z 1099.854,A 0.000,B 0.000,C 90.000,E1 189.726} C_DIS
LIN {X 0.072,Y -483.757,Z 1099.847,A 0.000,B 0.000,C 90.000,E1 188.454} C_DIS
LIN {X 0.116,Y -490.253,Z 1099.839,A 0.000,B 0.000,C 90.000,E1 187.068} C_DIS
LIN {X -0.050,Y -497.299,Z 1099.831,A 0.000,B 0.000,C 90.000,E1 185.568} C_DIS
LIN {X 0.093,Y -504.869,Z 1099.822,A 0.000,B 0.000,C 90.000,E1 183.898} C_DIS
LIN {X -0.097,Y -511.035,Z 1099.814,A 0.000,B 0.000,C 90.000,E1 182.579} C_DIS
LIN {X -0.024,Y -519.278,Z 1099.804,A 0.000,B 0.000,C 90.000,E1 180.802} C_DIS
LIN {X -0.021,Y -526.842,Z 1099.796,A 0.000,B 0.000,C 90.000,E1 179.198} C_DIS
LIN {X 0.147,Y -534.368,Z 1099.787,A 0.000,B 0.000,C 90.000,E1 177.593} C_DIS
LIN {X -0.085,Y -540.459,Z 1099.780,A 0.000,B 0.000,C 90.000,E1 176.331} C_DIS
LIN {X 0.073,Y -545.824,Z 1099.773,A 0.000,B 0.000,C 90.000,E1 175.179} C_DIS
LIN {X 0.065,Y -551.793,Z 1099.766,A 0.000,B 0.000,C 90.000,E1 173.913} C_DIS
LIN {X -0.029,Y -558.425,Z 1099.759,A 0.000,B 0.000,C 90.000,E1 172.527} C_DIS
LIN {X -0.011,Y -564.983,Z 1099.751,A 0.000,B 0.000,C 90.000,E1 171.141} C_DIS
LIN {X -0.216,Y -570.739,Z 1099.744,A 0.000,B 0.000,C 90.000,E1 169.926} C_DIS
LIN {X -0.241,Y -576.313,Z 1099.737,A 0.000,B 0.000,C 90.000,E1 168.701} C_DIS
LIN {X 0.051,Y -581.104,Z 1099.731,A 0.000,B 0.000,C 90.000,E1 167.589} C_DIS
LIN {X -0.029,Y -585.722,Z 1099.725,A 0.000,B 0.000,C 90.000,E1 166.520} C_DIS
LIN {X 0.075,Y -591.214,Z 1099.718,A 0.000,B 0.000,C 90.000,E1 165.172} C_DIS
LIN {X -0.159,Y -596.301,Z 1099.710,A 0.000,B 0.000,C 90.000,E1 163.866} C_DIS
LIN {X 0.149,Y -600.077,Z 1099.704,A 0.000,B 0.000,C 90.000,E1 162.779} C_DIS
LIN {X -0.239,Y -603.675,Z 1099.699,A 0.000,B 0.000,C 90.000,E1 161.764} C_DIS
LIN {X 0.178,Y -606.993,Z 1099.693,A 0.000,B 0.000,C 90.000,E1 160.678} C_DIS
LIN {X 0.067,Y -610.176,Z 1099.687,A 0.000,B 0.000,C 90.000,E1 159.645} C_DIS
LIN {X 0.173,Y -613.949,Z 1099.680,A 0.000,B 0.000,C 90.000,E1 158.337} C_DIS
LIN {X 0.121,Y -617.501,Z 1099.673,A 0.000,B 0.000,C 90.000,E1 157.050} C_DIS
LIN {X -0.205,Y -620.959,Z 1099.665,A 0.000,B 0.000,C 90.000,E1 155.793} C_DIS
LIN {X 0.091,Y -624.923,Z 1099.657,A 0.000,B 0.000,C 90.000,E1 154.229} C_DIS
LIN {X 0.134,Y -627.456,Z 1099.651,A 0.000,B 0.000,C 90.000,E1 153.204} C_DIS
LIN {X -0.027,Y -630.363,Z 1099.644,A 0.000,B 0.000,C 90.000,E1 151.948} C_DIS
LIN {X 0.121,Y -633.184,Z 1099.637,A 0.000,B 0.000,C 90.000,E1 150.667} C_DIS
LIN {X 0.065,Y -635.906,Z 1099.630,A 0.000,B 0.000,C 90.000,E1 149.410} C_DIS
LIN {X 0.007,Y -638.033,Z 1099.625,A 0.000,B 0.000,C 90.000,E1 148.408} C_DIS
LIN {X -0.176,Y -640.529,Z 1099.618,A 0.000,B 0.000,C 90.000,E1 147.168} C_DIS
LIN {X 0.221,Y -642.935,Z 1099.611,A 0.000,B 0.000,C 90.000,E1 145.881} C_DIS
LIN {X 0.008,Y -645.690,Z 1099.602,A 0.000,B 0.000,C 90.000,E1 144.402} C_DIS
LIN {X -0.154,Y -648.393,Z 1099.594,A 0.000,B 0.000,C 90.000,E1 142.924} C_DIS
LIN {X 0.084,Y -650.659,Z 1099.587,A 0.000,B 0.000,C 90.000,E1 141.662} C_DIS
LIN {X -0.098,Y -653.450,Z 1099.579,A 0.000,B 0.000,C 90.000,E1 140.194} C_DIS
LIN {X 0.150,Y -656.832,Z 1099.569,A 0.000,B 0.000,C 90.000,E1 138.447} C_DIS
LIN {X -0.013,Y -660.297,Z 1099.560,A 0.000,B 0.000,C 90.000,E1 136.743} C_DIS
LIN {X 0.337,Y -665.109,Z 1099.547,A 0.000,B 0.000,C 90.000,E1 134.514} C_DIS
LIN {X -0.121,Y -669.812,Z 1099.537,A 0.000,B 0.000,C 90.000,E1 132.609} C_DIS
LIN {X 0.004,Y -674.050,Z 1099.527,A 0.000,B 0.000,C 90.000,E1 130.906} C_DIS
LIN {X -0.248,Y -677.602,Z 1099.519,A 0.000,B 0.000,C 90.000,E1 129.483} C_DIS
LIN {X -0.300,Y -681.941,Z 1099.510,A 0.000,B 0.000,C 90.000,E1 127.810} C_DIS
LIN {X 0.093,Y -685.038,Z 1099.503,A 0.000,B 0.000,C 90.000,E1 126.583} C_DIS
LIN {X -0.055,Y -687.377,Z 1099.498,A 0.000,B 0.000,C 90.000,E1 125.644} C_DIS
LIN {X -0.210,Y -689.117,Z 1099.494,A 0.000,B 0.000,C 90.000,E1 124.945} C_DIS
LIN {X 0.221,Y -690.842,Z 1099.490,A 0.000,B 0.000,C 90.000,E1 124.199} C_DIS
LIN {X -0.010,Y -694.352,Z 1099.482,A 0.000,B 0.000,C 90.000,E1 122.801} C_DIS
LIN {X 0.372,Y -697.118,Z 1099.476,A 0.000,B 0.000,C 90.000,E1 121.592} C_DIS
LIN {X 0.187,Y -699.156,Z 1099.470,A 0.000,B 0.000,C 90.000,E1 120.669} C_DIS
LIN {X 0.032,Y -700.875,Z 1099.465,A 0.000,B 0.000,C 90.000,E1 119.745} C_DIS
LIN {X -0.102,Y -702.334,Z 1099.460,A 0.000,B 0.000,C 90.000,E1 118.821} C_DIS
LIN {X 0.115,Y -703.265,Z 1099.456,A 0.000,B 0.000,C 90.000,E1 118.103} C_DIS
LIN {X -0.002,Y -704.154,Z 1099.451,A 0.000,B 0.000,C 90.000,E1 117.180} C_DIS
LIN {X -0.170,Y -705.255,Z 1099.443,A 0.000,B 0.000,C 90.000,E1 115.796} C_DIS
LIN {X 0.062,Y -705.567,Z 1099.439,A 0.000,B 0.000,C 90.000,E1 115.079} C_DIS
LIN {X -0.297,Y -705.577,Z 1099.437,A 0.000,B 0.000,C 90.000,E1 114.643} C_DIS
LIN {X -0.009,Y -704.981,Z 1099.434,A 0.000,B 0.000,C 90.000,E1 114.155} C_DIS
LIN {X 0.280,Y -704.552,Z 1099.433,A 0.000,B 0.000,C 90.000,E1 113.898} C_DIS
LIN {X 0.062,Y -702.243,Z 1099.430,A 0.000,B 0.000,C 90.000,E1 113.334} C_DIS
LIN {X 0.200,Y -701.477,Z 1099.429,A 0.000,B 0.000,C 90.000,E1 113.206} C_DIS
LIN {X -0.177,Y -697.490,Z 1099.427,A 0.000,B 0.000,C 90.000,E1 112.770} C_DIS
LIN {X -0.048,Y -696.147,Z 1099.426,A 0.000,B 0.000,C 90.000,E1 112.642} C_DIS
LIN {X 0.080,Y -693.967,Z 1099.425,A 0.000,B 0.000,C 90.000,E1 112.514} C_DIS
LIN {X 0.118,Y -686.763,Z 1099.423,A 0.000,B 0.000,C 90.000,E1 112.206} C_DIS
LIN {X 0.006,Y -684.583,Z 1099.423,A 0.000,B 0.000,C 90.000,E1 112.153} C_DIS
LIN {X 0.286,Y -676.329,Z 1099.422,A 0.000,B 0.000,C 90.000,E1 112.025} C_DIS
LIN {X 0.208,Y -604.336,Z 1099.422,A 0.000,B 0.000,C 90.000,E1 112.025} C_DIS
LIN {X 0.236,Y -600.859,Z 1099.422,A 0.000,B 0.000,C 90.000,E1 111.844} C_DIS
LIN {X -0.011,Y -595.132,Z 1099.419,A 0.000,B 0.000,C 90.000,E1 111.461} C_DIS
LIN {X 0.109,Y -577.321,Z 1099.411,A 0.000,B 0.000,C 90.000,E1 109.939} C_DIS
LIN {X 0.084,Y -574.495,Z 1099.410,A 0.000,B 0.000,C 90.000,E1 109.704} C_DIS
LIN {X -0.090,Y -568.419,Z 1099.407,A 0.000,B 0.000,C 90.000,E1 109.268} C_DIS
LIN {X 0.225,Y -560.099,Z 1099.404,A 0.000,B 0.000,C 90.000,E1 108.725} C_DIS
LIN {X 0.108,Y -553.751,Z 1099.402,A 0.000,B 0.000,C 90.000,E1 108.362} C_DIS
LIN {X -0.088,Y -550.229,Z 1099.401,A 0.000,B 0.000,C 90.000,E1 108.127} C_DIS
LIN {X 0.083,Y -549.642,Z 1099.400,A 0.000,B 0.000,C 90.000,E1 108.055} C_DIS
LIN {X 0.134,Y -548.390,Z 1099.399,A 0.000,B 0.000,C 90.000,E1 107.873} C_DIS
LIN {X 0.092,Y -548.374,Z 1099.399,A 0.000,B 0.000,C 90.000,E1 107.873} C_DIS
LIN {X 0.055,Y -548.059,Z 1099.398,A 0.000,B 0.000,C 90.000,E1 107.583} C_DIS
LIN {X 0.092,Y -548.395,Z 1099.393,A 0.000,B 0.000,C 90.000,E1 106.677} C_DIS
LIN {X -0.084,Y -549.493,Z 1099.383,A 0.000,B 0.000,C 90.000,E1 105.009} C_DIS
LIN {X -0.040,Y -551.502,Z 1099.369,A 0.000,B 0.000,C 90.000,E1 102.479} C_DIS
LIN {X -0.291,Y -553.332,Z 1099.359,A 0.000,B 0.000,C 90.000,E1 100.546} C_DIS
LIN {X -0.061,Y -555.350,Z 1099.348,A 0.000,B 0.000,C 90.000,E1 98.568} C_DIS
LIN {X -0.002,Y -557.070,Z 1099.338,A 0.000,B 0.000,C 90.000,E1 96.891} C_DIS
LIN {X -0.100,Y -558.553,Z 1099.331,A 0.000,B 0.000,C 90.000,E1 95.511} C_DIS
LIN {X -0.246,Y -559.548,Z 1099.324,A 0.000,B 0.000,C 90.000,E1 94.416} C_DIS
LIN {X 0.047,Y -560.153,Z 1099.320,A 0.000,B 0.000,C 90.000,E1 93.555} C_DIS
LIN {X 0.067,Y -561.187,Z 1099.311,A 0.000,B 0.000,C 90.000,E1 91.892} C_DIS
LIN {X 0.008,Y -561.899,Z 1099.303,A 0.000,B 0.000,C 90.000,E1 90.516} C_DIS
LIN {X 0.150,Y -562.821,Z 1099.292,A 0.000,B 0.000,C 90.000,E1 88.568} C_DIS
LIN {X 0.217,Y -563.559,Z 1099.283,A 0.000,B 0.000,C 90.000,E1 86.906} C_DIS
LIN {X -0.235,Y -564.252,Z 1099.274,A 0.000,B 0.000,C 90.000,E1 85.298} C_DIS
LIN {X -0.060,Y -564.832,Z 1099.265,A 0.000,B 0.000,C 90.000,E1 83.628} C_DIS
LIN {X -0.052,Y -565.251,Z 1099.259,A 0.000,B 0.000,C 90.000,E1 82.527} C_DIS
LIN {X 0.223,Y -565.776,Z 1099.249,A 0.000,B 0.000,C 90.000,E1 80.849} C_DIS
LIN {X 0.039,Y -566.481,Z 1099.240,A 0.000,B 0.000,C 90.000,E1 79.218} C_DIS
LIN {X -0.141,Y -567.258,Z 1099.231,A 0.000,B 0.000,C 90.000,E1 77.589} C_DIS
LIN {X -0.241,Y -567.923,Z 1099.223,A 0.000,B 0.000,C 90.000,E1 76.228} C_DIS
LIN {X 0.028,Y -569.068,Z 1099.213,A 0.000,B 0.000,C 90.000,E1 74.283} C_DIS
LIN {X -0.292,Y -570.702,Z 1099.201,A 0.000,B 0.000,C 90.000,E1 72.127} C_DIS
LIN {X -0.018,Y -572.282,Z 1099.190,A 0.000,B 0.000,C 90.000,E1 70.188} C_DIS
LIN {X 0.129,Y -573.746,Z 1099.181,A 0.000,B 0.000,C 90.000,E1 68.539} C_DIS
LIN {X -0.015,Y -575.172,Z 1099.172,A 0.000,B 0.000,C 90.000,E1 66.922} C_DIS
LIN {X -0.043,Y -576.752,Z 1099.161,A 0.000,B 0.000,C 90.000,E1 65.025} C_DIS
LIN {X -0.034,Y -578.063,Z 1099.151,A 0.000,B 0.000,C 90.000,E1 63.127} C_DIS
LIN {X -0.118,Y -579.135,Z 1099.142,A 0.000,B 0.000,C 90.000,E1 61.513} C_DIS
LIN {X 0.095,Y -579.832,Z 1099.136,A 0.000,B 0.000,C 90.000,E1 60.411} C_DIS
LIN {X 0.111,Y -580.684,Z 1099.127,A 0.000,B 0.000,C 90.000,E1 58.791} C_DIS
LIN {X -0.005,Y -581.441,Z 1099.119,A 0.000,B 0.000,C 90.000,E1 57.454} C_DIS
LIN {X 0.196,Y -582.100,Z 1099.112,A 0.000,B 0.000,C 90.000,E1 56.087} C_DIS
LIN {X -0.092,Y -582.512,Z 1099.107,A 0.000,B 0.000,C 90.000,E1 55.308} C_DIS
LIN {X -0.177,Y -583.204,Z 1099.098,A 0.000,B 0.000,C 90.000,E1 53.703} C_DIS
LIN {X -0.094,Y -583.638,Z 1099.091,A 0.000,B 0.000,C 90.000,E1 52.351} C_DIS
LIN {X 0.169,Y -583.913,Z 1099.085,A 0.000,B 0.000,C 90.000,E1 51.251} C_DIS
LIN {X -0.013,Y -583.827,Z 1099.079,A 0.000,B 0.000,C 90.000,E1 50.194} C_DIS
LIN {X -0.016,Y -583.637,Z 1099.071,A 0.000,B 0.000,C 90.000,E1 48.852} C_DIS
LIN {X -0.204,Y -583.340,Z 1099.065,A 0.000,B 0.000,C 90.000,E1 47.796} C_DIS
LIN {X -0.271,Y -582.801,Z 1099.058,A 0.000,B 0.000,C 90.000,E1 46.458} C_DIS
LIN {X 0.060,Y -582.100,Z 1099.051,A 0.000,B 0.000,C 90.000,E1 45.081} C_DIS
LIN {X -0.177,Y -581.304,Z 1099.045,A 0.000,B 0.000,C 90.000,E1 44.028} C_DIS
LIN {X -0.008,Y -580.180,Z 1099.039,A 0.000,B 0.000,C 90.000,E1 42.933} C_DIS
LIN {X 0.146,Y -578.933,Z 1099.033,A 0.000,B 0.000,C 90.000,E1 41.838} C_DIS
LIN {X -0.257,Y -577.811,Z 1099.028,A 0.000,B 0.000,C 90.000,E1 41.067} C_DIS
LIN {X -0.003,Y -575.657,Z 1099.021,A 0.000,B 0.000,C 90.000,E1 39.688} C_DIS
LIN {X -0.221,Y -573.639,Z 1099.015,A 0.000,B 0.000,C 90.000,E1 38.624} C_DIS
LIN {X -0.099,Y -571.246,Z 1099.008,A 0.000,B 0.000,C 90.000,E1 37.523} C_DIS
LIN {X -0.151,Y -569.172,Z 1099.004,A 0.000,B 0.000,C 90.000,E1 36.710} C_DIS
LIN {X -0.107,Y -566.727,Z 1098.999,A 0.000,B 0.000,C 90.000,E1 35.884} C_DIS
LIN {X 0.131,Y -564.958,Z 1098.996,A 0.000,B 0.000,C 90.000,E1 35.311} C_DIS
LIN {X 0.032,Y -562.953,Z 1098.993,A 0.000,B 0.000,C 90.000,E1 34.771} C_DIS
LIN {X 0.240,Y -560.809,Z 1098.990,A 0.000,B 0.000,C 90.000,E1 34.199} C_DIS
LIN {X 0.314,Y -557.858,Z 1098.986,A 0.000,B 0.000,C 90.000,E1 33.499} C_DIS
LIN {X 0.123,Y -553.414,Z 1098.981,A 0.000,B 0.000,C 90.000,E1 32.546} C_DIS
LIN {X -0.004,Y -549.186,Z 1098.976,A 0.000,B 0.000,C 90.000,E1 31.720} C_DIS
LIN {X 0.159,Y -543.932,Z 1098.971,A 0.000,B 0.000,C 90.000,E1 30.718} C_DIS
LIN {X 0.250,Y -539.801,Z 1098.967,A 0.000,B 0.000,C 90.000,E1 30.001} C_DIS
LIN {X -0.023,Y -536.384,Z 1098.964,A 0.000,B 0.000,C 90.000,E1 29.461} C_DIS
LIN {X 0.146,Y -532.673,Z 1098.961,A 0.000,B 0.000,C 90.000,E1 28.871} C_DIS
LIN {X 0.135,Y -527.712,Z 1098.957,A 0.000,B 0.000,C 90.000,E1 28.153} C_DIS
LIN {X -0.160,Y -522.267,Z 1098.953,A 0.000,B 0.000,C 90.000,E1 27.462} C_DIS
LIN {X -0.260,Y -516.361,Z 1098.948,A 0.000,B 0.000,C 90.000,E1 26.744} C_DIS
LIN {X 0.219,Y -511.265,Z 1098.945,A 0.000,B 0.000,C 90.000,E1 26.104} C_DIS
LIN {X -0.221,Y -501.984,Z 1098.940,A 0.000,B 0.000,C 90.000,E1 25.155} C_DIS
LIN {X 0.128,Y -492.664,Z 1098.934,A 0.000,B 0.000,C 90.000,E1 24.155} C_DIS
LIN {X 0.152,Y -485.465,Z 1098.931,A 0.000,B 0.000,C 90.000,E1 23.462} C_DIS
LIN {X -0.158,Y -476.842,Z 1098.926,A 0.000,B 0.000,C 90.000,E1 22.695} C_DIS
LIN {X -0.001,Y -466.550,Z 1098.921,A 0.000,B 0.000,C 90.000,E1 21.770} C_DIS
LIN {X 0.128,Y -448.827,Z 1098.912,A 0.000,B 0.000,C 90.000,E1 20.194} C_DIS
LIN {X -0.209,Y -432.673,Z 1098.904,A 0.000,B 0.000,C 90.000,E1 18.725} C_DIS
LIN {X 0.108,Y -419.795,Z 1098.896,A 0.000,B 0.000,C 90.000,E1 17.347} C_DIS
LIN {X 0.004,Y -408.737,Z 1098.889,A 0.000,B 0.000,C 90.000,E1 16.079} C_DIS
LIN {X -0.127,Y -402.111,Z 1098.885,A 0.000,B 0.000,C 90.000,E1 15.245} C_DIS
LIN {X -0.055,Y -397.325,Z 1098.881,A 0.000,B 0.000,C 90.000,E1 14.537} C_DIS
LIN {X -0.020,Y -396.290,Z 1098.880,A 0.000,B 0.000,C 90.000,E1 14.356} C_DIS
LIN {X 0.050,Y -394.678,Z 1098.878,A 0.000,B 0.000,C 90.000,E1 14.008} C_DIS
LIN {X 0.181,Y -394.070,Z 1098.877,A 0.000,B 0.000,C 90.000,E1 13.828} C_DIS
LIN {X 0.095,Y -392.539,Z 1098.874,A 0.000,B 0.000,C 90.000,E1 13.300} C_DIS
LIN {X 0.070,Y -392.059,Z 1098.871,A 0.000,B 0.000,C 90.000,E1 12.771} C_DIS
LIN {X 0.128,Y -392.285,Z 1098.868,A 0.000,B 0.000,C 90.000,E1 12.187} C_DIS
LIN {X 0.117,Y -393.051,Z 1098.864,A 0.000,B 0.000,C 90.000,E1 11.478} C_DIS
LIN {X -0.008,Y -396.111,Z 1098.854,A 0.000,B 0.000,C 90.000,E1 9.726} C_DIS
LIN {X 0.162,Y -401.498,Z 1098.840,A 0.000,B 0.000,C 90.000,E1 7.239} C_DIS
LIN {X 0.093,Y -403.212,Z 1098.837,A 0.000,B 0.000,C 90.000,E1 6.549} C_DIS
LIN {X 0.040,Y -406.581,Z 1098.829,A 0.000,B 0.000,C 90.000,E1 5.163} C_DIS
LIN {X 0.014,Y -409.273,Z 1098.825,A 0.000,B 0.000,C 90.000,E1 4.473} C_DIS
LIN {X -0.184,Y -411.865,Z 1098.823,A 0.000,B 0.000,C 90.000,E1 4.069} C_DIS
LIN {X 0.195,Y -415.874,Z 1098.820,A 0.000,B 0.000,C 90.000,E1 3.612} C_DIS
LIN {X -0.022,Y -419.951,Z 1098.818,A 0.000,B 0.000,C 90.000,E1 3.326} C_DIS
LIN {X -0.120,Y -441.256,Z 1098.810,A 0.000,B 0.000,C 90.000,E1 1.892} C_DIS
LIN {X -0.052,Y -464.322,Z 1098.802,A 0.000,B 0.000,C 90.000,E1 0.401} C_DIS
LIN {X -0.212,Y -475.531,Z 1098.798,A 0.000,B 0.000,C 90.000,E1 359.714} C_DIS
LIN {X -0.068,Y -486.774,Z 1098.794,A 0.000,B 0.000,C 90.000,E1 358.969} C_DIS
LIN {X -0.132,Y -496.289,Z 1098.791,A 0.000,B 0.000,C 90.000,E1 358.339} C_DIS
LIN {X 0.092,Y -503.830,Z 1098.788,A 0.000,B 0.000,C 90.000,E1 357.764} C_DIS
LIN {X 0.069,Y -511.229,Z 1098.785,A 0.000,B 0.000,C 90.000,E1 357.192} C_DIS
LIN {X -0.152,Y -517.089,Z 1098.782,A 0.000,B 0.000,C 90.000,E1 356.731} C_DIS
LIN {X -0.194,Y -524.108,Z 1098.778,A 0.000,B 0.000,C 90.000,E1 356.102} C_DIS
LIN {X -0.087,Y -528.212,Z 1098.776,A 0.000,B 0.000,C 90.000,E1 355.698} C_DIS
LIN {X -0.030,Y -534.603,Z 1098.772,A 0.000,B 0.000,C 90.000,E1 355.008} C_DIS
LIN {X -0.052,Y -540.451,Z 1098.768,A 0.000,B 0.000,C 90.000,E1 354.318} C_DIS
LIN {X -0.245,Y -545.828,Z 1098.765,A 0.000,B 0.000,C 90.000,E1 353.628} C_DIS
LIN {X -0.140,Y -549.818,Z 1098.761,A 0.000,B 0.000,C 90.000,E1 353.053} C_DIS
LIN {X 0.066,Y -553.447,Z 1098.758,A 0.000,B 0.000,C 90.000,E1 352.470} C_DIS
LIN {X -0.023,Y -557.443,Z 1098.754,A 0.000,B 0.000,C 90.000,E1 351.781} C_DIS
LIN {X 0.001,Y -561.011,Z 1098.750,A 0.000,B 0.000,C 90.000,E1 351.084} C_DIS
LIN {X 0.058,Y -564.277,Z 1098.747,A 0.000,B 0.000,C 90.000,E1 350.387} C_DIS
LIN {X 0.003,Y -567.867,Z 1098.742,A 0.000,B 0.000,C 90.000,E1 349.567} C_DIS
LIN {X -0.125,Y -571.209,Z 1098.738,A 0.000,B 0.000,C 90.000,E1 348.757} C_DIS
LIN {X 0.087,Y -575.237,Z 1098.731,A 0.000,B 0.000,C 90.000,E1 347.645} C_DIS
LIN {X 0.006,Y -579.862,Z 1098.724,A 0.000,B 0.000,C 90.000,E1 346.297} C_DIS
LIN {X -0.039,Y -584.981,Z 1098.715,A 0.000,B 0.000,C 90.000,E1 344.685} C_DIS
LIN {X 0.190,Y -588.971,Z 1098.708,A 0.000,B 0.000,C 90.000,E1 343.323} C_DIS
LIN {X -0.344,Y -592.095,Z 1098.702,A 0.000,B 0.000,C 90.000,E1 342.308} C_DIS
LIN {X -0.094,Y -595.076,Z 1098.696,A 0.000,B 0.000,C 90.000,E1 341.221} C_DIS
LIN {X -0.061,Y -597.079,Z 1098.691,A 0.000,B 0.000,C 90.000,E1 340.423} C_DIS
LIN {X 0.168,Y -600.089,Z 1098.684,A 0.000,B 0.000,C 90.000,E1 339.082} C_DIS
LIN {X 0.182,Y -602.244,Z 1098.678,A 0.000,B 0.000,C 90.000,E1 338.028} C_DIS
LIN {X 0.228,Y -604.103,Z 1098.672,A 0.000,B 0.000,C 90.000,E1 336.975} C_DIS
LIN {X 0.296,Y -605.596,Z 1098.666,A 0.000,B 0.000,C 90.000,E1 335.921} C_DIS
LIN {X -0.178,Y -607.005,Z 1098.661,A 0.000,B 0.000,C 90.000,E1 334.921} C_DIS
LIN {X 0.121,Y -608.332,Z 1098.653,A 0.000,B 0.000,C 90.000,E1 333.589} C_DIS
LIN {X -0.018,Y -608.891,Z 1098.649,A 0.000,B 0.000,C 90.000,E1 332.820} C_DIS
LIN {X 0.133,Y -609.333,Z 1098.645,A 0.000,B 0.000,C 90.000,E1 332.025} C_DIS
LIN {X -0.040,Y -609.673,Z 1098.639,A 0.000,B 0.000,C 90.000,E1 331.001} C_DIS
LIN {X 0.170,Y -609.702,Z 1098.636,A 0.000,B 0.000,C 90.000,E1 330.461} C_DIS
LIN {X -0.233,Y -609.221,Z 1098.630,A 0.000,B 0.000,C 90.000,E1 329.459} C_DIS
LIN {X -0.068,Y -608.471,Z 1098.626,A 0.000,B 0.000,C 90.000,E1 328.663} C_DIS
LIN {X 0.085,Y -607.425,Z 1098.622,A 0.000,B 0.000,C 90.000,E1 327.867} C_DIS
LIN {X -0.224,Y -606.729,Z 1098.619,A 0.000,B 0.000,C 90.000,E1 327.375} C_DIS
LIN {X 0.163,Y -604.571,Z 1098.613,A 0.000,B 0.000,C 90.000,E1 326.294} C_DIS
LIN {X 0.011,Y -602.314,Z 1098.607,A 0.000,B 0.000,C 90.000,E1 325.261} C_DIS
LIN {X -0.066,Y -599.356,Z 1098.600,A 0.000,B 0.000,C 90.000,E1 323.956} C_DIS
LIN {X -0.296,Y -596.817,Z 1098.594,A 0.000,B 0.000,C 90.000,E1 322.924} C_DIS
LIN {X 0.377,Y -593.792,Z 1098.587,A 0.000,B 0.000,C 90.000,E1 321.537} C_DIS
LIN {X -0.091,Y -590.016,Z 1098.578,A 0.000,B 0.000,C 90.000,E1 319.989} C_DIS
LIN {X -0.003,Y -586.866,Z 1098.570,A 0.000,B 0.000,C 90.000,E1 318.647} C_DIS
LIN {X 0.317,Y -585.411,Z 1098.567,A 0.000,B 0.000,C 90.000,E1 318.081} C_DIS
LIN {X -0.023,Y -583.072,Z 1098.563,A 0.000,B 0.000,C 90.000,E1 317.310} C_DIS
LIN {X 0.013,Y -580.232,Z 1098.558,A 0.000,B 0.000,C 90.000,E1 316.500} C_DIS
LIN {X -0.105,Y -578.315,Z 1098.555,A 0.000,B 0.000,C 90.000,E1 315.972} C_DIS
LIN {X 0.025,Y -575.540,Z 1098.552,A 0.000,B 0.000,C 90.000,E1 315.283} C_DIS
LIN {X 0.124,Y -572.510,Z 1098.548,A 0.000,B 0.000,C 90.000,E1 314.595} C_DIS
LIN {X 0.092,Y -570.818,Z 1098.546,A 0.000,B 0.000,C 90.000,E1 314.190} C_DIS
LIN {X -0.215,Y -564.402,Z 1098.538,A 0.000,B 0.000,C 90.000,E1 312.852} C_DIS
LIN {X -0.058,Y -561.600,Z 1098.535,A 0.000,B 0.000,C 90.000,E1 312.285} C_DIS
LIN {X -0.072,Y -557.855,Z 1098.531,A 0.000,B 0.000,C 90.000,E1 311.595} C_DIS
LIN {X 0.095,Y -552.921,Z 1098.526,A 0.000,B 0.000,C 90.000,E1 310.744} C_DIS
LIN {X 0.216,Y -549.386,Z 1098.523,A 0.000,B 0.000,C 90.000,E1 310.172} C_DIS
LIN {X -0.104,Y -546.166,Z 1098.520,A 0.000,B 0.000,C 90.000,E1 309.644} C_DIS
LIN {X 0.163,Y -542.676,Z 1098.516,A 0.000,B 0.000,C 90.000,E1 308.910} C_DIS
LIN {X -0.047,Y -540.849,Z 1098.514,A 0.000,B 0.000,C 90.000,E1 308.508} C_DIS
LIN {X -0.022,Y -539.948,Z 1098.512,A 0.000,B 0.000,C 90.000,E1 308.222} C_DIS
LIN {X -0.001,Y -539.214,Z 1098.511,A 0.000,B 0.000,C 90.000,E1 307.935} C_DIS
LIN {X 0.017,Y -538.337,Z 1098.509,A 0.000,B 0.000,C 90.000,E1 307.649} C_DIS
LIN {X 0.032,Y -537.729,Z 1098.508,A 0.000,B 0.000,C 90.000,E1 307.363} C_DIS
LIN {X 0.045,Y -537.394,Z 1098.506,A 0.000,B 0.000,C 90.000,E1 307.076} C_DIS
LIN {X 0.065,Y -536.274,Z 1098.503,A 0.000,B 0.000,C 90.000,E1 306.503} C_DIS
LIN {X -0.228,Y -535.122,Z 1098.497,A 0.000,B 0.000,C 90.000,E1 305.391} C_DIS
LIN {X 0.228,Y -534.665,Z 1098.489,A 0.000,B 0.000,C 90.000,E1 303.913} C_DIS
LIN {X -0.077,Y -534.705,Z 1098.485,A 0.000,B 0.000,C 90.000,E1 303.372} C_DIS
LIN {X -0.108,Y -535.708,Z 1098.469,A 0.000,B 0.000,C 90.000,E1 300.512} C_DIS
LIN {X 0.221,Y -536.353,Z 1098.463,A 0.000,B 0.000,C 90.000,E1 299.333} C_DIS
LIN {X -0.165,Y -536.951,Z 1098.457,A 0.000,B 0.000,C 90.000,E1 298.231} C_DIS
LIN {X -0.160,Y -537.980,Z 1098.446,A 0.000,B 0.000,C 90.000,E1 296.232} C_DIS
LIN {X 0.171,Y -538.554,Z 1098.438,A 0.000,B 0.000,C 90.000,E1 294.771} C_DIS
LIN {X -0.207,Y -538.984,Z 1098.430,A 0.000,B 0.000,C 90.000,E1 293.387} C_DIS
LIN {X -0.066,Y -539.404,Z 1098.420,A 0.000,B 0.000,C 90.000,E1 291.663} C_DIS
LIN {X -0.137,Y -539.605,Z 1098.412,A 0.000,B 0.000,C 90.000,E1 290.248} C_DIS
LIN {X 0.070,Y -539.556,Z 1098.406,A 0.000,B 0.000,C 90.000,E1 289.087} C_DIS
LIN {X -0.194,Y -539.325,Z 1098.398,A 0.000,B 0.000,C 90.000,E1 287.692} C_DIS
LIN {X -0.112,Y -539.039,Z 1098.390,A 0.000,B 0.000,C 90.000,E1 286.260} C_DIS
LIN {X -0.037,Y -538.483,Z 1098.382,A 0.000,B 0.000,C 90.000,E1 284.828} C_DIS
LIN {X -0.114,Y -537.889,Z 1098.375,A 0.000,B 0.000,C 90.000,E1 283.411} C_DIS
LIN {X -0.194,Y -536.904,Z 1098.363,A 0.000,B 0.000,C 90.000,E1 281.422} C_DIS
LIN {X 0.052,Y -536.331,Z 1098.357,A 0.000,B 0.000,C 90.000,E1 280.254} C_DIS
LIN {X -0.170,Y -535.351,Z 1098.346,A 0.000,B 0.000,C 90.000,E1 278.276} C_DIS
LIN {X -0.041,Y -534.374,Z 1098.335,A 0.000,B 0.000,C 90.000,E1 276.258} C_DIS
LIN {X 0.028,Y -533.554,Z 1098.325,A 0.000,B 0.000,C 90.000,E1 274.531} C_DIS
LIN {X 0.023,Y -532.610,Z 1098.314,A 0.000,B 0.000,C 90.000,E1 272.522} C_DIS
LIN {X -0.026,Y -531.711,Z 1098.303,A 0.000,B 0.000,C 90.000,E1 270.516} C_DIS
LIN {X -0.097,Y -530.804,Z 1098.293,A 0.000,B 0.000,C 90.000,E1 268.797} C_DIS
LIN {X -0.159,Y -529.991,Z 1098.285,A 0.000,B 0.000,C 90.000,E1 267.364} C_DIS
LIN {X -0.203,Y -529.103,Z 1098.277,A 0.000,B 0.000,C 90.000,E1 265.927} C_DIS
LIN {X 0.252,Y -528.396,Z 1098.271,A 0.000,B 0.000,C 90.000,E1 264.723} C_DIS
LIN {X 0.210,Y -527.508,Z 1098.264,A 0.000,B 0.000,C 90.000,E1 263.571} C_DIS
LIN {X 0.201,Y -526.658,Z 1098.260,A 0.000,B 0.000,C 90.000,E1 262.704} C_DIS
LIN {X 0.153,Y -524.834,Z 1098.250,A 0.000,B 0.000,C 90.000,E1 260.971} C_DIS
LIN {X 0.250,Y -522.814,Z 1098.239,A 0.000,B 0.000,C 90.000,E1 258.926} C_DIS
LIN {X -0.207,Y -520.822,Z 1098.227,A 0.000,B 0.000,C 90.000,E1 256.937} C_DIS
LIN {X -0.097,Y -519.146,Z 1098.218,A 0.000,B 0.000,C 90.000,E1 255.172} C_DIS
LIN {X 0.241,Y -517.354,Z 1098.208,A 0.000,B 0.000,C 90.000,E1 253.378} C_DIS
LIN {X 0.176,Y -515.139,Z 1098.196,A 0.000,B 0.000,C 90.000,E1 251.329} C_DIS
LIN {X -0.147,Y -513.839,Z 1098.190,A 0.000,B 0.000,C 90.000,E1 250.188} C_DIS
LIN {X 0.030,Y -511.498,Z 1098.178,A 0.000,B 0.000,C 90.000,E1 248.103} C_DIS
LIN {X 0.119,Y -509.678,Z 1098.170,A 0.000,B 0.000,C 90.000,E1 246.613} C_DIS
LIN {X 0.012,Y -506.983,Z 1098.160,A 0.000,B 0.000,C 90.000,E1 244.845} C_DIS
LIN {X 0.133,Y -505.046,Z 1098.154,A 0.000,B 0.000,C 90.000,E1 243.640} C_DIS
LIN {X 0.139,Y -502.091,Z 1098.144,A 0.000,B 0.000,C 90.000,E1 241.847} C_DIS
LIN {X 0.259,Y -499.614,Z 1098.135,A 0.000,B 0.000,C 90.000,E1 240.333} C_DIS
LIN {X -0.096,Y -497.000,Z 1098.127,A 0.000,B 0.000,C 90.000,E1 238.869} C_DIS
LIN {X 0.033,Y -493.799,Z 1098.117,A 0.000,B 0.000,C 90.000,E1 237.041} C_DIS
LIN {X 0.104,Y -491.041,Z 1098.109,A 0.000,B 0.000,C 90.000,E1 235.515} C_DIS
LIN {X -0.115,Y -488.729,Z 1098.102,A 0.000,B 0.000,C 90.000,E1 234.322} C_DIS
LIN {X 0.143,Y -485.754,Z 1098.093,A 0.000,B 0.000,C 90.000,E1 232.763} C_DIS
LIN {X 0.130,Y -483.335,Z 1098.086,A 0.000,B 0.000,C 90.000,E1 231.537} C_DIS
LIN {X -0.111,Y -481.409,Z 1098.081,A 0.000,B 0.000,C 90.000,E1 230.642} C_DIS
LIN {X -0.089,Y -478.305,Z 1098.073,A 0.000,B 0.000,C 90.000,E1 229.094} C_DIS
LIN {X -0.195,Y -473.440,Z 1098.059,A 0.000,B 0.000,C 90.000,E1 226.620} C_DIS
LIN {X 0.029,Y -470.038,Z 1098.048,A 0.000,B 0.000,C 90.000,E1 224.717} C_DIS
LIN {X 0.025,Y -467.768,Z 1098.042,A 0.000,B 0.000,C 90.000,E1 223.461} C_DIS
LIN {X -0.199,Y -464.214,Z 1098.031,A 0.000,B 0.000,C 90.000,E1 221.595} C_DIS
LIN {X -0.200,Y -461.330,Z 1098.022,A 0.000,B 0.000,C 90.000,E1 220.011} C_DIS
LIN {X 0.096,Y -458.524,Z 1098.013,A 0.000,B 0.000,C 90.000,E1 218.382} C_DIS
LIN {X 0.233,Y -454.244,Z 1097.999,A 0.000,B 0.000,C 90.000,E1 215.804} C_DIS
LIN {X 0.005,Y -450.572,Z 1097.987,A 0.000,B 0.000,C 90.000,E1 213.579} C_DIS
LIN {X -0.042,Y -448.583,Z 1097.979,A 0.000,B 0.000,C 90.000,E1 212.291} C_DIS
LIN {X 0.021,Y -445.441,Z 1097.969,A 0.000,B 0.000,C 90.000,E1 210.335} C_DIS
LIN {X 0.163,Y -442.688,Z 1097.958,A 0.000,B 0.000,C 90.000,E1 208.359} C_DIS
LIN {X 0.157,Y -438.556,Z 1097.939,A 0.000,B 0.000,C 90.000,E1 205.079} C_DIS
LIN {X 0.170,Y -436.736,Z 1097.927,A 0.000,B 0.000,C 90.000,E1 202.770} C_DIS
LIN {X 0.073,Y -436.539,Z 1097.919,A 0.000,B 0.000,C 90.000,E1 201.461} C_DIS
LIN {X -0.021,Y -437.098,Z 1097.914,A 0.000,B 0.000,C 90.000,E1 200.482} C_DIS
LIN {X 0.056,Y -437.890,Z 1097.910,A 0.000,B 0.000,C 90.000,E1 199.812} C_DIS
LIN {X 0.140,Y -439.024,Z 1097.906,A 0.000,B 0.000,C 90.000,E1 199.141} C_DIS
LIN {X -0.069,Y -441.425,Z 1097.901,A 0.000,B 0.000,C 90.000,E1 198.181} C_DIS
LIN {X -0.249,Y -444.433,Z 1097.896,A 0.000,B 0.000,C 90.000,E1 197.221} C_DIS
LIN {X 0.068,Y -450.532,Z 1097.886,A 0.000,B 0.000,C 90.000,E1 195.552} C_DIS
LIN {X -0.152,Y -458.554,Z 1097.876,A 0.000,B 0.000,C 90.000,E1 193.647} C_DIS
LIN {X 0.042,Y -467.001,Z 1097.865,A 0.000,B 0.000,C 90.000,E1 191.715} C_DIS
LIN {X 0.200,Y -477.358,Z 1097.853,A 0.000,B 0.000,C 90.000,E1 189.500} C_DIS
LIN {X 0.071,Y -483.322,Z 1097.846,A 0.000,B 0.000,C 90.000,E1 188.276} C_DIS
LIN {X 0.103,Y -489.881,Z 1097.838,A 0.000,B 0.000,C 90.000,E1 186.891} C_DIS
LIN {X -0.078,Y -497.007,Z 1097.830,A 0.000,B 0.000,C 90.000,E1 185.391} C_DIS
LIN {X 0.012,Y -504.647,Z 1097.821,A 0.000,B 0.000,C 90.000,E1 183.726} C_DIS
LIN {X -0.179,Y -510.873,Z 1097.813,A 0.000,B 0.000,C 90.000,E1 182.407} C_DIS
LIN {X 0.023,Y -516.389,Z 1097.807,A 0.000,B 0.000,C 90.000,E1 181.203} C_DIS
LIN {X 0.064,Y -521.277,Z 1097.801,A 0.000,B 0.000,C 90.000,E1 180.172} C_DIS
LIN {X -0.142,Y -528.223,Z 1097.793,A 0.000,B 0.000,C 90.000,E1 178.740} C_DIS
LIN {X 0.051,Y -535.830,Z 1097.784,A 0.000,B 0.000,C 90.000,E1 177.135} C_DIS
LIN {X -0.091,Y -544.672,Z 1097.774,A 0.000,B 0.000,C 90.000,E1 175.298} C_DIS
LIN {X 0.126,Y -550.008,Z 1097.768,A 0.000,B 0.000,C 90.000,E1 174.147} C_DIS
LIN {X -0.255,Y -557.354,Z 1097.759,A 0.000,B 0.000,C 90.000,E1 172.648} C_DIS
LIN {X 0.133,Y -564.599,Z 1097.751,A 0.000,B 0.000,C 90.000,E1 171.084} C_DIS
LIN {X -0.219,Y -571.025,Z 1097.743,A 0.000,B 0.000,C 90.000,E1 169.746} C_DIS
LIN {X 0.127,Y -575.366,Z 1097.738,A 0.000,B 0.000,C 90.000,E1 168.757} C_DIS
LIN {X 0.079,Y -579.617,Z 1097.732,A 0.000,B 0.000,C 90.000,E1 167.813} C_DIS
LIN {X 0.090,Y -585.413,Z 1097.725,A 0.000,B 0.000,C 90.000,E1 166.464} C_DIS
LIN {X 0.186,Y -590.967,Z 1097.717,A 0.000,B 0.000,C 90.000,E1 165.117} C_DIS
LIN {X -0.324,Y -595.099,Z 1097.712,A 0.000,B 0.000,C 90.000,E1 164.102} C_DIS
LIN {X -0.033,Y -598.941,Z 1097.706,A 0.000,B 0.000,C 90.000,E1 163.015} C_DIS
LIN {X 0.139,Y -602.588,Z 1097.700,A 0.000,B 0.000,C 90.000,E1 161.945} C_DIS
LIN {X -0.029,Y -605.982,Z 1097.694,A 0.000,B 0.000,C 90.000,E1 160.913} C_DIS
LIN {X -0.151,Y -609.220,Z 1097.688,A 0.000,B 0.000,C 90.000,E1 159.880} C_DIS
LIN {X -0.281,Y -613.049,Z 1097.681,A 0.000,B 0.000,C 90.000,E1 158.592} C_DIS
LIN {X 0.188,Y -617.376,Z 1097.672,A 0.000,B 0.000,C 90.000,E1 156.997} C_DIS
LIN {X 0.118,Y -620.146,Z 1097.667,A 0.000,B 0.000,C 90.000,E1 155.973} C_DIS
LIN {X -0.156,Y -624.155,Z 1097.658,A 0.000,B 0.000,C 90.000,E1 154.460} C_DIS
LIN {X -0.100,Y -627.327,Z 1097.651,A 0.000,B 0.000,C 90.000,E1 153.179} C_DIS
LIN {X 0.007,Y -630.250,Z 1097.644,A 0.000,B 0.000,C 90.000,E1 151.897} C_DIS
LIN {X -0.093,Y -633.072,Z 1097.637,A 0.000,B 0.000,C 90.000,E1 150.639} C_DIS
LIN {X -0.101,Y -636.320,Z 1097.628,A 0.000,B 0.000,C 90.000,E1 149.125} C_DIS
LIN {X -0.149,Y -638.429,Z 1097.623,A 0.000,B 0.000,C 90.000,E1 148.122} C_DIS
LIN {X -0.275,Y -641.387,Z 1097.615,A 0.000,B 0.000,C 90.000,E1 146.628} C_DIS
LIN {X 0.130,Y -643.760,Z 1097.608,A 0.000,B 0.000,C 90.000,E1 145.341} C_DIS
LIN {X -0.075,Y -646.519,Z 1097.599,A 0.000,B 0.000,C 90.000,E1 143.863} C_DIS
LIN {X 0.080,Y -649.720,Z 1097.590,A 0.000,B 0.000,C 90.000,E1 142.110} C_DIS
LIN {X 0.322,Y -652.949,Z 1097.580,A 0.000,B 0.000,C 90.000,E1 140.356} C_DIS
LIN {X 0.082,Y -656.801,Z 1097.569,A 0.000,B 0.000,C 90.000,E1 138.405} C_DIS
LIN {X -0.095,Y -660.286,Z 1097.559,A 0.000,B 0.000,C 90.000,E1 136.701} C_DIS
LIN {X -0.230,Y -665.123,Z 1097.547,A 0.000,B 0.000,C 90.000,E1 134.514} C_DIS
LIN {X 0.250,Y -669.261,Z 1097.538,A 0.000,B 0.000,C 90.000,E1 132.771} C_DIS
LIN {X -0.059,Y -674.112,Z 1097.527,A 0.000,B 0.000,C 90.000,E1 130.862} C_DIS
LIN {X 0.131,Y -677.654,Z 1097.519,A 0.000,B 0.000,C 90.000,E1 129.402} C_DIS
LIN {X 0.079,Y -681.997,Z 1097.510,A 0.000,B 0.000,C 90.000,E1 127.729} C_DIS
LIN {X 0.065,Y -685.113,Z 1097.503,A 0.000,B 0.000,C 90.000,E1 126.537} C_DIS
LIN {X -0.075,Y -687.422,Z 1097.498,A 0.000,B 0.000,C 90.000,E1 125.598} C_DIS
LIN {X 0.002,Y -690.357,Z 1097.491,A 0.000,B 0.000,C 90.000,E1 124.405} C_DIS
LIN {X -0.009,Y -694.415,Z 1097.482,A 0.000,B 0.000,C 90.000,E1 122.752} C_DIS
LIN {X -0.213,Y -697.166,Z 1097.475,A 0.000,B 0.000,C 90.000,E1 121.592} C_DIS
LIN {X -0.400,Y -699.205,Z 1097.470,A 0.000,B 0.000,C 90.000,E1 120.669} C_DIS
LIN {X 0.401,Y -700.914,Z 1097.465,A 0.000,B 0.000,C 90.000,E1 119.667} C_DIS
LIN {X 0.263,Y -702.355,Z 1097.460,A 0.000,B 0.000,C 90.000,E1 118.743} C_DIS
LIN {X -0.192,Y -703.467,Z 1097.455,A 0.000,B 0.000,C 90.000,E1 117.847} C_DIS
LIN {X 0.320,Y -704.264,Z 1097.449,A 0.000,B 0.000,C 90.000,E1 116.873} C_DIS
LIN {X 0.181,Y -705.203,Z 1097.443,A 0.000,B 0.000,C 90.000,E1 115.720} C_DIS
LIN {X 0.109,Y -705.500,Z 1097.439,A 0.000,B 0.000,C 90.000,E1 115.027} C_DIS
LIN {X -0.247,Y -705.484,Z 1097.437,A 0.000,B 0.000,C 90.000,E1 114.591} C_DIS
LIN {X 0.330,Y -704.858,Z 1097.434,A 0.000,B 0.000,C 90.000,E1 114.079} C_DIS
LIN {X -0.313,Y -704.322,Z 1097.433,A 0.000,B 0.000,C 90.000,E1 113.898} C_DIS
LIN {X 0.253,Y -702.525,Z 1097.430,A 0.000,B 0.000,C 90.000,E1 113.387} C_DIS
LIN {X 0.392,Y -701.928,Z 1097.429,A 0.000,B 0.000,C 90.000,E1 113.259} C_DIS
LIN {X 0.013,Y -698.080,Z 1097.427,A 0.000,B 0.000,C 90.000,E1 112.823} C_DIS
LIN {X -0.125,Y -697.000,Z 1097.426,A 0.000,B 0.000,C 90.000,E1 112.717} C_DIS
LIN {X 0.004,Y -695.390,Z 1097.426,A 0.000,B 0.000,C 90.000,E1 112.589} C_DIS
LIN {X -0.118,Y -689.361,Z 1097.424,A 0.000,B 0.000,C 90.000,E1 112.333} C_DIS
LIN {X -0.256,Y -685.931,Z 1097.423,A 0.000,B 0.000,C 90.000,E1 112.206} C_DIS
LIN {X -0.281,Y -683.071,Z 1097.423,A 0.000,B 0.000,C 90.000,E1 112.153} C_DIS
LIN {X 0.234,Y -676.374,Z 1097.422,A 0.000,B 0.000,C 90.000,E1 112.025} C_DIS
LIN {X 0.161,Y -604.401,Z 1097.422,A 0.000,B 0.000,C 90.000,E1 112.025} C_DIS
LIN {X 0.000,Y -600.664,Z 1097.421,A 0.000,B 0.000,C 90.000,E1 111.844} C_DIS
LIN {X 0.019,Y -596.191,Z 1097.420,A 0.000,B 0.000,C 90.000,E1 111.535} C_DIS
LIN {X 0.207,Y -575.994,Z 1097.410,A 0.000,B 0.000,C 90.000,E1 109.812} C_DIS
LIN {X 0.302,Y -571.390,Z 1097.408,A 0.000,B 0.000,C 90.000,E1 109.450} C_DIS
LIN {X -0.077,Y -568.439,Z 1097.407,A 0.000,B 0.000,C 90.000,E1 109.268} C_DIS
LIN {X 0.235,Y -560.108,Z 1097.404,A 0.000,B 0.000,C 90.000,E1 108.725} C_DIS
LIN {X 0.118,Y -553.751,Z 1097.402,A 0.000,B 0.000,C 90.000,E1 108.362} C_DIS
LIN {X 0.230,Y -549.704,Z 1097.401,A 0.000,B 0.000,C 90.000,E1 108.055} C_DIS
LIN {X 0.149,Y -548.354,Z 1097.399,A 0.000,B 0.000,C 90.000,E1 107.873} C_DIS
LIN {X 0.107,Y -548.328,Z 1097.399,A 0.000,B 0.000,C 90.000,E1 107.873} C_DIS
LIN {X 0.103,Y -547.987,Z 1097.397,A 0.000,B 0.000,C 90.000,E1 107.457} C_DIS
LIN {X 0.292,Y -548.322,Z 1097.393,A 0.000,B 0.000,C 90.000,E1 106.677} C_DIS
LIN {X 0.115,Y -549.411,Z 1097.384,A 0.000,B 0.000,C 90.000,E1 105.009} C_DIS
LIN {X 0.156,Y -551.392,Z 1097.370,A 0.000,B 0.000,C 90.000,E1 102.479} C_DIS
LIN {X 0.206,Y -552.690,Z 1097.362,A 0.000,B 0.000,C 90.000,E1 101.074} C_DIS
LIN {X 0.008,Y -554.971,Z 1097.349,A 0.000,B 0.000,C 90.000,E1 98.859} C_DIS
LIN {X 0.064,Y -556.704,Z 1097.340,A 0.000,B 0.000,C 90.000,E1 97.182} C_DIS
LIN {X 0.021,Y -558.217,Z 1097.332,A 0.000,B 0.000,C 90.000,E1 95.796} C_DIS
LIN {X -0.135,Y -559.272,Z 1097.326,A 0.000,B 0.000,C 90.000,E1 94.702} C_DIS
LIN {X 0.238,Y -560.109,Z 1097.320,A 0.000,B 0.000,C 90.000,E1 93.555} C_DIS
LIN {X 0.258,Y -561.115,Z 1097.311,A 0.000,B 0.000,C 90.000,E1 91.892} C_DIS
LIN {X 0.197,Y -561.829,Z 1097.303,A 0.000,B 0.000,C 90.000,E1 90.516} C_DIS
LIN {X 0.237,Y -562.591,Z 1097.294,A 0.000,B 0.000,C 90.000,E1 88.854} C_DIS
LIN {X 0.099,Y -563.108,Z 1097.288,A 0.000,B 0.000,C 90.000,E1 87.764} C_DIS
LIN {X 0.174,Y -563.786,Z 1097.278,A 0.000,B 0.000,C 90.000,E1 86.102} C_DIS
LIN {X 0.192,Y -564.352,Z 1097.271,A 0.000,B 0.000,C 90.000,E1 84.723} C_DIS
LIN {X -0.033,Y -565.033,Z 1097.260,A 0.000,B 0.000,C 90.000,E1 82.818} C_DIS
LIN {X 0.233,Y -565.575,Z 1097.251,A 0.000,B 0.000,C 90.000,E1 81.141} C_DIS
LIN {X 0.215,Y -566.382,Z 1097.240,A 0.000,B 0.000,C 90.000,E1 79.218} C_DIS
LIN {X 0.207,Y -567.274,Z 1097.230,A 0.000,B 0.000,C 90.000,E1 77.297} C_DIS
LIN {X 0.224,Y -568.441,Z 1097.217,A 0.000,B 0.000,C 90.000,E1 75.102} C_DIS
LIN {X -0.090,Y -570.154,Z 1097.204,A 0.000,B 0.000,C 90.000,E1 72.670} C_DIS
LIN {X -0.182,Y -571.465,Z 1097.195,A 0.000,B 0.000,C 90.000,E1 71.040} C_DIS
LIN {X 0.309,Y -573.167,Z 1097.184,A 0.000,B 0.000,C 90.000,E1 69.082} C_DIS
LIN {X 0.105,Y -574.335,Z 1097.176,A 0.000,B 0.000,C 90.000,E1 67.741} C_DIS
LIN {X -0.014,Y -575.245,Z 1097.170,A 0.000,B 0.000,C 90.000,E1 66.666} C_DIS
LIN {X -0.128,Y -576.623,Z 1097.161,A 0.000,B 0.000,C 90.000,E1 65.049} C_DIS
LIN {X 0.122,Y -577.927,Z 1097.151,A 0.000,B 0.000,C 90.000,E1 63.127} C_DIS
LIN {X 0.036,Y -578.979,Z 1097.142,A 0.000,B 0.000,C 90.000,E1 61.513} C_DIS
LIN {X -0.258,Y -579.676,Z 1097.136,A 0.000,B 0.000,C 90.000,E1 60.461} C_DIS
LIN {X 0.115,Y -580.672,Z 1097.125,A 0.000,B 0.000,C 90.000,E1 58.535} C_DIS
LIN {X -0.010,Y -581.429,Z 1097.118,A 0.000,B 0.000,C 90.000,E1 57.199} C_DIS
LIN {X -0.125,Y -582.249,Z 1097.109,A 0.000,B 0.000,C 90.000,E1 55.595} C_DIS
LIN {X -0.218,Y -582.915,Z 1097.100,A 0.000,B 0.000,C 90.000,E1 53.989} C_DIS
LIN {X -0.319,Y -583.302,Z 1097.094,A 0.000,B 0.000,C 90.000,E1 52.924} C_DIS
LIN {X 0.301,Y -583.700,Z 1097.085,A 0.000,B 0.000,C 90.000,E1 51.251} C_DIS
LIN {X 0.293,Y -583.539,Z 1097.078,A 0.000,B 0.000,C 90.000,E1 49.908} C_DIS
LIN {X -0.158,Y -583.310,Z 1097.070,A 0.000,B 0.000,C 90.000,E1 48.609} C_DIS
LIN {X 0.212,Y -582.842,Z 1097.063,A 0.000,B 0.000,C 90.000,E1 47.229} C_DIS
LIN {X 0.139,Y -582.247,Z 1097.055,A 0.000,B 0.000,C 90.000,E1 45.891} C_DIS
LIN {X -0.095,Y -581.630,Z 1097.049,A 0.000,B 0.000,C 90.000,E1 44.838} C_DIS
LIN {X -0.072,Y -580.970,Z 1097.045,A 0.000,B 0.000,C 90.000,E1 44.028} C_DIS
LIN {X -0.178,Y -579.533,Z 1097.037,A 0.000,B 0.000,C 90.000,E1 42.690} C_DIS
LIN {X 0.243,Y -578.576,Z 1097.033,A 0.000,B 0.000,C 90.000,E1 41.838} C_DIS
LIN {X -0.165,Y -577.425,Z 1097.028,A 0.000,B 0.000,C 90.000,E1 41.067} C_DIS
LIN {X -0.287,Y -575.235,Z 1097.021,A 0.000,B 0.000,C 90.000,E1 39.725} C_DIS
LIN {X -0.142,Y -573.185,Z 1097.015,A 0.000,B 0.000,C 90.000,E1 38.624} C_DIS
LIN {X -0.306,Y -572.022,Z 1097.011,A 0.000,B 0.000,C 90.000,E1 38.096} C_DIS
LIN {X 0.241,Y -569.410,Z 1097.005,A 0.000,B 0.000,C 90.000,E1 36.950} C_DIS
LIN {X -0.169,Y -567.043,Z 1097.001,A 0.000,B 0.000,C 90.000,E1 36.171} C_DIS
LIN {X 0.188,Y -564.375,Z 1096.996,A 0.000,B 0.000,C 90.000,E1 35.311} C_DIS
LIN {X 0.084,Y -562.393,Z 1096.993,A 0.000,B 0.000,C 90.000,E1 34.771} C_DIS
LIN {X 0.381,Y -559.003,Z 1096.989,A 0.000,B 0.000,C 90.000,E1 33.913} C_DIS
LIN {X 0.321,Y -555.328,Z 1096.984,A 0.000,B 0.000,C 90.000,E1 33.086} C_DIS
LIN {X 0.038,Y -552.055,Z 1096.980,A 0.000,B 0.000,C 90.000,E1 32.418} C_DIS
LIN {X 0.023,Y -548.462,Z 1096.976,A 0.000,B 0.000,C 90.000,E1 31.720} C_DIS
LIN {X 0.175,Y -543.186,Z 1096.971,A 0.000,B 0.000,C 90.000,E1 30.718} C_DIS
LIN {X 0.260,Y -539.070,Z 1096.967,A 0.000,B 0.000,C 90.000,E1 30.001} C_DIS
LIN {X -0.157,Y -534.691,Z 1096.963,A 0.000,B 0.000,C 90.000,E1 29.333} C_DIS
LIN {X 0.145,Y -531.870,Z 1096.961,A 0.000,B 0.000,C 90.000,E1 28.871} C_DIS
LIN {X 0.028,Y -527.858,Z 1096.957,A 0.000,B 0.000,C 90.000,E1 28.309} C_DIS
LIN {X -0.177,Y -521.380,Z 1096.953,A 0.000,B 0.000,C 90.000,E1 27.462} C_DIS
LIN {X -0.284,Y -515.400,Z 1096.948,A 0.000,B 0.000,C 90.000,E1 26.744} C_DIS
LIN {X -0.098,Y -511.612,Z 1096.946,A 0.000,B 0.000,C 90.000,E1 26.283} C_DIS
LIN {X 0.012,Y -502.515,Z 1096.941,A 0.000,B 0.000,C 90.000,E1 25.283} C_DIS
LIN {X -0.237,Y -491.725,Z 1096.934,A 0.000,B 0.000,C 90.000,E1 24.207} C_DIS
LIN {X 0.074,Y -480.783,Z 1096.929,A 0.000,B 0.000,C 90.000,E1 23.131} C_DIS
LIN {X -0.146,Y -472.238,Z 1096.924,A 0.000,B 0.000,C 90.000,E1 22.386} C_DIS
LIN {X 0.084,Y -466.364,Z 1096.922,A 0.000,B 0.000,C 90.000,E1 21.844} C_DIS
LIN {X -0.035,Y -450.113,Z 1096.914,A 0.000,B 0.000,C 90.000,E1 20.429} C_DIS
LIN {X 0.201,Y -433.998,Z 1096.905,A 0.000,B 0.000,C 90.000,E1 18.906} C_DIS
LIN {X 0.124,Y -419.799,Z 1096.897,A 0.000,B 0.000,C 90.000,E1 17.457} C_DIS
LIN {X -0.126,Y -407.676,Z 1096.889,A 0.000,B 0.000,C 90.000,E1 16.079} C_DIS
LIN {X 0.016,Y -400.138,Z 1096.884,A 0.000,B 0.000,C 90.000,E1 15.064} C_DIS
LIN {X 0.031,Y -397.035,Z 1096.881,A 0.000,B 0.000,C 90.000,E1 14.592} C_DIS
LIN {X 0.065,Y -394.990,Z 1096.879,A 0.000,B 0.000,C 90.000,E1 14.189} C_DIS
LIN {X 0.096,Y -394.155,Z 1096.878,A 0.000,B 0.000,C 90.000,E1 14.008} C_DIS
LIN {X -0.072,Y -392.596,Z 1096.875,A 0.000,B 0.000,C 90.000,E1 13.480} C_DIS
LIN {X -0.007,Y -392.136,Z 1096.872,A 0.000,B 0.000,C 90.000,E1 12.939} C_DIS
LIN {X -0.055,Y -392.223,Z 1096.870,A 0.000,B 0.000,C 90.000,E1 12.591} C_DIS
LIN {X -0.103,Y -392.367,Z 1096.868,A 0.000,B 0.000,C 90.000,E1 12.243} C_DIS
LIN {X -0.115,Y -393.125,Z 1096.864,A 0.000,B 0.000,C 90.000,E1 11.535} C_DIS
LIN {X 0.061,Y -398.317,Z 1096.848,A 0.000,B 0.000,C 90.000,E1 8.681} C_DIS
LIN {X -0.146,Y -403.205,Z 1096.837,A 0.000,B 0.000,C 90.000,E1 6.606} C_DIS
LIN {X 0.202,Y -406.521,Z 1096.829,A 0.000,B 0.000,C 90.000,E1 5.163} C_DIS
LIN {X 0.170,Y -407.685,Z 1096.827,A 0.000,B 0.000,C 90.000,E1 4.821} C_DIS
LIN {X 0.173,Y -409.831,Z 1096.824,A 0.000,B 0.000,C 90.000,E1 4.302} C_DIS
LIN {X -0.061,Y -411.863,Z 1096.822,A 0.000,B 0.000,C 90.000,E1 4.012} C_DIS
LIN {X -0.116,Y -414.563,Z 1096.821,A 0.000,B 0.000,C 90.000,E1 3.726} C_DIS
LIN {X 0.039,Y -416.117,Z 1096.820,A 0.000,B 0.000,C 90.000,E1 3.555} C_DIS
LIN {X -0.196,Y -421.941,Z 1096.817,A 0.000,B 0.000,C 90.000,E1 3.151} C_DIS
LIN {X 0.136,Y -439.967,Z 1096.811,A 0.000,B 0.000,C 90.000,E1 1.892} C_DIS
LIN {X 0.017,Y -459.741,Z 1096.804,A 0.000,B 0.000,C 90.000,E1 0.630} C_DIS
LIN {X 0.180,Y -473.154,Z 1096.799,A 0.000,B 0.000,C 90.000,E1 359.771} C_DIS
LIN {X -0.154,Y -484.504,Z 1096.795,A 0.000,B 0.000,C 90.000,E1 359.083} C_DIS
LIN {X -0.106,Y -495.606,Z 1096.791,A 0.000,B 0.000,C 90.000,E1 358.339} C_DIS
LIN {X 0.096,Y -503.311,Z 1096.788,A 0.000,B 0.000,C 90.000,E1 357.764} C_DIS
LIN {X 0.068,Y -510.789,Z 1096.785,A 0.000,B 0.000,C 90.000,E1 357.192} C_DIS
LIN {X -0.155,Y -516.714,Z 1096.782,A 0.000,B 0.000,C 90.000,E1 356.731} C_DIS
LIN {X -0.123,Y -523.733,Z 1096.778,A 0.000,B 0.000,C 90.000,E1 356.102} C_DIS
LIN {X -0.109,Y -529.069,Z 1096.775,A 0.000,B 0.000,C 90.000,E1 355.584} C_DIS
LIN {X 0.153,Y -534.219,Z 1096.772,A 0.000,B 0.000,C 90.000,E1 355.008} C_DIS
LIN {X -0.137,Y -541.274,Z 1096.768,A 0.000,B 0.000,C 90.000,E1 354.204} C_DIS
LIN {X -0.064,Y -545.596,Z 1096.765,A 0.000,B 0.000,C 90.000,E1 353.628} C_DIS
LIN {X 0.081,Y -549.623,Z 1096.761,A 0.000,B 0.000,C 90.000,E1 353.053} C_DIS
LIN {X 0.071,Y -554.096,Z 1096.758,A 0.000,B 0.000,C 90.000,E1 352.356} C_DIS
LIN {X 0.068,Y -558.078,Z 1096.754,A 0.000,B 0.000,C 90.000,E1 351.659} C_DIS
LIN {X 0.014,Y -561.635,Z 1096.750,A 0.000,B 0.000,C 90.000,E1 350.971} C_DIS
LIN {X -0.236,Y -564.262,Z 1096.747,A 0.000,B 0.000,C 90.000,E1 350.443} C_DIS
LIN {X 0.164,Y -567.888,Z 1096.742,A 0.000,B 0.000,C 90.000,E1 349.577} C_DIS
LIN {X -0.233,Y -572.312,Z 1096.736,A 0.000,B 0.000,C 90.000,E1 348.522} C_DIS
LIN {X -0.005,Y -576.292,Z 1096.730,A 0.000,B 0.000,C 90.000,E1 347.409} C_DIS
LIN {X -0.067,Y -580.882,Z 1096.723,A 0.000,B 0.000,C 90.000,E1 346.061} C_DIS
LIN {X 0.084,Y -585.195,Z 1096.715,A 0.000,B 0.000,C 90.000,E1 344.700} C_DIS
LIN {X -0.091,Y -589.219,Z 1096.708,A 0.000,B 0.000,C 90.000,E1 343.378} C_DIS
LIN {X -0.187,Y -593.147,Z 1096.700,A 0.000,B 0.000,C 90.000,E1 342.054} C_DIS
LIN {X 0.200,Y -595.400,Z 1096.696,A 0.000,B 0.000,C 90.000,E1 341.221} C_DIS
LIN {X 0.237,Y -597.419,Z 1096.691,A 0.000,B 0.000,C 90.000,E1 340.423} C_DIS
LIN {X -0.087,Y -600.471,Z 1096.684,A 0.000,B 0.000,C 90.000,E1 339.135} C_DIS
LIN {X -0.290,Y -602.626,Z 1096.678,A 0.000,B 0.000,C 90.000,E1 338.103} C_DIS
LIN {X -0.245,Y -604.523,Z 1096.672,A 0.000,B 0.000,C 90.000,E1 337.050} C_DIS
